//		E_WorkingStates.NOTIFY_LOADING_OUTBOUND:
//			ton_timeout.PT	:= T#1S;
//			///////////////there is no tote in working position/////////////
//			IF NOT(roller_inbound.photo_sensor[0].Q OR roller_inbound.photo_sensor[1].Q OR photo_sensor_tote_detection.Q OR roller_outbound.photo_sensor.Q) THEN
//				IF sInstanceName='working1' THEN
//					subData.Topic	:= E_Topics.LOADING_BEGIN_OUTBOUND_WOKING1;
//					GVL.PubSubService.Publish(topic:=E_Topics.LOADING_BEGIN_OUTBOUND_WOKING1,data:= subData);				
//				END_IF
//				IF sInstanceName='working2' THEN
//					subData.Topic	:= E_Topics.LOADING_BEGIN_OUTBOUND_WOKING2;
//					GVL.PubSubService.Publish(topic:=E_Topics.LOADING_BEGIN_OUTBOUND_WOKING2,data:= subData);				
//				END_IF
//				eStates	:= E_WorkingStates.WAIT_NEW_TOTE;
//			END_IF	
//			///////////////there is a tote in working position/////////////
//			IF NOT roller_inbound.photo_sensor[0].Q AND roller_inbound.photo_sensor[1].Q AND photo_sensor_tote_detection.Q AND NOT roller_outbound.photo_sensor.Q THEN
//				eStates	:= E_WorkingStates.BAG_OPEN_DOWN;
//			END_IF					
			
		E_WorkingStates.WAIT_NEW_TOTE:	
			///////////////there is a tote in working position/////////////
			IF NOT roller_inbound.photo_sensor[0].Q AND roller_inbound.photo_sensor[1].Q AND photo_sensor_tote_detection.Q AND NOT roller_outbound.photo_sensor.Q THEN
				eStates	:= E_WorkingStates.BAG_OPEN_DOWN;
			END_IF			
		/////////////////////////abort inbound command from app///////////////////
			IF xAbortInbound THEN
				xAbortInbound	:= FALSE;
				tote_status	:= ToteStatus.VACANT;
				M_load	:= TRUE;
				eStates	:= E_WorkingStates.IDLE;				
			ELSE
				tote_status	:= ToteStatus.AWAITING_INBOUND_AVAILABILITY;
			END_IF
		//////////////////////////normal process///////////////////////
			IF sInstanceName='working1' THEN
				IF xBeginInbound AND GVL.fb_loading.valve_left_door.retracted THEN
					xBeginInbound	:=FALSE;
					eStates	:= E_WorkingStates.WAIT_MUTE_SENSOR_ON;
				END_IF					
			END_IF
			IF sInstanceName='working2' THEN
				IF xBeginInbound AND GVL.fb_loading.valve_right_door.retracted THEN
					xBeginInbound	:=FALSE;
					eStates	:= E_WorkingStates.WAIT_MUTE_SENSOR_ON;
				END_IF					
			END_IF
		/////////////////////////////while in stopping/////////////////////			
			IF  THIS^.eState = ePMLState_Stopping THEN
				IF sInstanceName='working1' THEN//publish to loading for loading might be not in stopping
					subData.Topic	:= E_Topics.LOADING_END_OUTBOUND_WOKING1;
					GVL.PubSubService.Publish(topic:=E_Topics.LOADING_END_OUTBOUND_WOKING1,data:= subData);				
				END_IF
				IF sInstanceName='working2' THEN
					subData.Topic	:= E_Topics.LOADING_END_OUTBOUND_WOKING2;
					GVL.PubSubService.Publish(topic:=E_Topics.LOADING_END_OUTBOUND_WOKING2,data:= subData);				
				END_IF
				M_load	:= TRUE;
				eStates	:= E_WorkingStates.IDLE;
			END_IF						
////////////////////////////////////////////////action/////////////////////////////////////////////
			
		E_WorkingStates.WAIT_MUTE_SENSOR_ON:	
			tote_status	:= ToteStatus.INBOUNDING;
			ton_timeout.PT	:= T#2S;	
			roller_inbound.roller.forward	:= TRUE;
			IF  roller_inbound.photo_sensor[0].Q THEN
				eStates	:= E_WorkingStates.WAIT_TOTE_DETECTION_ON;
			END_IF			
		E_WorkingStates.WAIT_TOTE_DETECTION_ON:
			roller_inbound.roller.forward	:= TRUE;
			IF photo_sensor_tote_detection.Q THEN
				eStates	:= E_WorkingStates.WAIT_MUTE_SENSOR_OFF;
			END_IF
		E_WorkingStates.WAIT_MUTE_SENSOR_OFF:
			roller_inbound.roller.forward	:= TRUE;
			IF NOT roller_inbound.photo_sensor[0].Q THEN
				eStates	:= E_WorkingStates.WAIT_LOAD_SENSOR_ON;
			END_IF
		E_WorkingStates.WAIT_LOAD_SENSOR_ON:
			roller_inbound.roller.forward	:= TRUE;
			IF roller_inbound.photo_sensor[1].Q THEN	
				roller_inbound.roller.forward	:= FALSE;
				eStates	:= E_WorkingStates.BAG_OPEN_DOWN;
			END_IF
		E_WorkingStates.BAG_OPEN_DOWN:
			st_mcAxis_lift.mcMoveAbsolute.Execute	:= TRUE;		
			st_mcAxis_lift.rActualPosSet	:= rPos_lift_down;
			st_mcAxis_lift.rVelocitySet	:= 250;
			IF st_mcAxis_lift.mcMoveAbsolute.Done THEN	
				eStates	:= E_WorkingStates.BAG_OPEN;
			END_IF		
		E_WorkingStates.BAG_OPEN:	
			ton_timeout.PT	:= T#3S;		
			st_mcAxis_bag.mcMoveAbsolute.Execute	:= TRUE;		
			st_mcAxis_bag.rActualPosSet	:= rPos_bag_opened;
			st_mcAxis_bag.rVelocitySet	:= 50;
			IF st_mcAxis_bag.mcMoveAbsolute.Done OR st_mcAxis_bag.bTouchTorque THEN			
				st_mcAxis_bag.mcMoveAbsolute.Execute	:= FALSE;
				eStates	:= E_WorkingStates.BAG_OPEN_DETECTION;
			END_IF	
		E_WorkingStates.BAG_OPEN_DETECTION:	
			IF ABS(st_mcAxis_bag.rActualPos-rPos_bag_opened)>5 THEN
				bagOpen_Status[0].bag_status	:= BagStatus.ERROR;
				bagOpen_Status[1].bag_status	:= BagStatus.ERROR;
				tote_status	:= ToteStatus.BAG_OPEN_FAILED;
				eStates	:= E_WorkingStates.DONE;
				RETURN;
			END_IF
			ton_timeout.PT	:= INT_TO_TIME(iDelay_sensor_detection);
			IF ton_timeout.Q THEN
				/////////////////////////////////////////////bag openner1/////////////////////////////////////////					
				FOR i:=0 TO 3 DO
					IF BagOpening_Detection[i] THEN
						bagOpen_Status[0].sensor_status	:=CONCAT(STR1:=bagOpen_Status[0].sensor_status,STR2:='1');
						bagOpen_Status[0].iCnt_sensor_detection	:=bagOpen_Status[0].iCnt_sensor_detection+1;
					ELSE
						bagOpen_Status[0].sensor_status	:=CONCAT(STR1:=bagOpen_Status[0].sensor_status,STR2:='0');
					END_IF
				END_FOR	
				IF bagOpen_Status[0].iCnt_sensor_detection>=iSensor_detection_setting[0] THEN
					bagOpen_Status[0].bag_status	:= BagStatus.OPENED;
					strLog_bagopen_detection	:= CONCAT(STR1:=bag_opening_status[0].sensor_status,STR2:='->OPENED;');
				ELSE
					bagOpen_Status[0].bag_status	:= BagStatus.ERROR;
					strLog_bagopen_detection	:= CONCAT(STR1:=bag_opening_status[0].sensor_status,STR2:='->ERROR;');
				END_IF			
				/////////////////////////////////////////////bag openner2/////////////////////////////////////////	
				FOR i:=4 TO 7 DO
					IF BagOpening_Detection[i] THEN
						bagOpen_Status[1].sensor_status	:=CONCAT(STR1:=bagOpen_Status[1].sensor_status,STR2:='1');
						bagOpen_Status[1].iCnt_sensor_detection	:=bagOpen_Status[1].iCnt_sensor_detection+1;
					ELSE
						bagOpen_Status[1].sensor_status	:=CONCAT(STR1:=bagOpen_Status[1].sensor_status,STR2:='0');
					END_IF
				END_FOR		
				IF bagOpen_Status[1].iCnt_sensor_detection>=iSensor_detection_setting[1] THEN
					bagOpen_Status[1].bag_status	:= BagStatus.OPENED;
					strLog_bagopen_detection	:= CONCAT(STR1:=bag_opening_status[1].sensor_status,STR2:='->OPENED');
				ELSE
					bagOpen_Status[1].bag_status	:= BagStatus.ERROR;
					strLog_bagopen_detection	:= CONCAT(STR1:=bag_opening_status[1].sensor_status,STR2:='->ERROR');
				END_IF				

	
				eStates	:= E_WorkingStates.TOTE_STATUS_DETECTION;	
			END_IF
		E_WorkingStates.TOTE_STATUS_DETECTION:
			IF bUsingOpenBag THEN
				IF bagOpen_Status[0].bag_status=BagStatus.OPENED AND bagOpen_Status[1].bag_status=BagStatus.OPENED THEN
					tote_status	:= ToteStatus.LOADED;
				ELSE
					tote_status	:= ToteStatus.BAG_OPEN_FAILED;
				END_IF
			ELSE
				tote_status	:= ToteStatus.LOADED;
			END_IF
			/////////////////////////////////////////writelog////////////////////////////////////////
			IF bagOpen_Status[0].bag_status=BagStatus.OPENED THEN
				strLog_bagopen_detection	:= CONCAT(STR1:=bagOpen_Status[0].sensor_status,STR2:='->OPENED;');
			ELSE	
				strLog_bagopen_detection	:= CONCAT(STR1:=bagOpen_Status[0].sensor_status,STR2:='->ERROR;');
			END_IF
			IF bagOpen_Status[1].bag_status=BagStatus.OPENED THEN
				strLog_bagopen_detection	:= CONCAT(STR1:=strLog_bagopen_detection,STR2:=bagOpen_Status[1].sensor_status);
				strLog_bagopen_detection	:= CONCAT(STR1:=strLog_bagopen_detection,STR2:='->OPENED;');
			ELSE	
				strLog_bagopen_detection	:= CONCAT(STR1:=strLog_bagopen_detection,STR2:=bagOpen_Status[1].sensor_status);
				strLog_bagopen_detection	:= CONCAT(STR1:=strLog_bagopen_detection,STR2:='->ERROR;');
			END_IF					
			eStates	:= E_WorkingStates.DONE;		
		E_WorkingStates.DONE:
			ADSLOGSTR(msgCtrlMask:= ADSLOG_MSGTYPE_LOG,msgFmtStr:=strLog_bagopen_detection,strArg:='');
			M_load	:= TRUE;
			eStates	:= E_WorkingStates.IDLE;
			

		
		
END_CASE
END_METHOD

METHOD M_mapping : BOOL
VAR_INPUT
END_VAR
IF sInstanceName='working1' THEN
	
	/////////////////////////////////////digital input-2024.5.25////////////////////////////////////////

	roller_inbound.roller.err(D:= G_IO.arDI[4].Ch[0],on_ms:=500,off_ms:=80);	
	roller_inbound.photo_sensor[0](D:= arIOLinkQualifier_Place1.CH[3].1,on_ms:=200,off_ms:=300);  //入口料框检测
	roller_inbound.photo_sensor[1](D:= arIOLinkQualifier_Place1.CH[3].0,on_ms:=100,off_ms:=100);  //X向到位感应
	
	roller_outbound.roller.err(D:= G_IO.arDI[4].Ch[1],on_ms:=500,off_ms:=80);	
	roller_outbound.photo_sensor(D:= arIOLinkQualifier_Place1.CH[4].0,on_ms:=100,off_ms:=80);   //Y向出料口感应

	roller_outbound_assist.roller.err(D:= G_IO.arDI[4].Ch[2],on_ms:=500,off_ms:=80);	
	EDM_KM            							:= G_IO.arDI[4].Ch[3];       //P24_sto反馈  
				  
	photo_sensor_tote_detection(D:= arIOLinkQualifier_Place1.CH[4].1,on_ms:=100,off_ms:=100);  //XY对角料框感应
		
	BagOpening_Detection[0]:= arIOLinkTx_Place1[7].	InputByte[1].0;
	BagOpening_Detection[1]:= arIOLinkTx_Place1[7].	InputByte[0].0;
	BagOpening_Detection[2]:= arIOLinkTx_Place1[7].	InputByte[1].1;
	BagOpening_Detection[3]:= arIOLinkTx_Place1[7].	InputByte[0].1;
	BagOpening_Detection[4]:= arIOLinkTx_Place1[7].	InputByte[1].2;
	BagOpening_Detection[5]:= arIOLinkTx_Place1[7].	InputByte[0].2;
	BagOpening_Detection[6]:= arIOLinkTx_Place1[7].	InputByte[1].3;
	BagOpening_Detection[7]:= arIOLinkTx_Place1[7].	InputByte[0].3;
		
	valve_lift.extended		:= arIOLinkQualifier_Place1.CH[0].1 AND arIOLinkQualifier_Place1.CH[1].1;
	valve_lift.retracted	:= arIOLinkQualifier_Place1.CH[2].1 AND arIOLinkQualifier_Place1.CH[2].0;
		
	(****************************axis_lift*******************************************************)
		
	st_mcAxis_lift.limit_sensor_positive:= arIOLinkQualifier_Place1.CH[5].0	 ;
	st_mcAxis_lift.limit_sensor_negative:= arIOLinkQualifier_Place1.CH[5].1  ;
	st_mcAxis_lift.limit_sensor_home	:= arIOLinkQualifier_Place1.CH[6].1  ;
		
		
		
		
	(****************************axis_bagopener***************************************************)
	st_mcAxis_bag.limit_sensor_positive:= 	arIOLinkTx_Place1[7].InputByte[0].4 ;
	st_mcAxis_bag.limit_sensor_negative:= 	arIOLinkTx_Place1[7].InputByte[0].5 ;
	//using software limit position for
		
		
		
		
		
	/////////////////////////////////////digital output-2024.5.25////////////////////////////////////////
	G_IO.arDO[6].Ch[0]	:= valve_lift.extend;
	G_IO.arDO[6].Ch[1]	:= valve_lift.retract;
		
	G_IO.arDO[4].Ch[2]	:= roller_inbound.roller.forward;
	G_IO.arDO[4].Ch[3]	:= roller_inbound.roller.backward;		
	G_IO.arDO[4].Ch[4]	:= roller_outbound.roller.backward;
	G_IO.arDO[4].Ch[5]	:= roller_outbound.roller.forward;		
	G_IO.arDO[4].Ch[6]	:= roller_outbound_assist.roller.forward;
	G_IO.arDO[4].Ch[7]	:= roller_outbound_assist.roller.backward;
			
	/////////////////////////////////////axis config////////////////////////////////////////
	mcAxis_lift
	(
		ZSN		:=   st_mcAxis_lift.limit_sensor_negative OR st_mcAxis_lift.xHoming, //TODO link to digital input
		ZSP		:=   st_mcAxis_lift.limit_sensor_positive  OR st_mcAxis_lift.xHoming, //TODO link to digital input
		IN_OUT	:= st_mcAxis_lift	, 
		AXIS	:= AxisRef_lift	, 
	);
	st_mcAxis_lift.bPosSensorShow	:= TRUE;
	st_mcAxis_lift.bNegSensorShow	:= TRUE;
	st_mcAxis_lift.bStopButtonShow	:= TRUE;
	st_mcAxis_lift.rMaxAcceleration	:= 50000;
	st_mcAxis_lift.rMaxDeceleration	:= 50000;
	st_mcAxis_lift.rMaxJerk			:= 500000;
	st_mcAxis_lift.rAcceleration	:= 2500;
	st_mcAxis_lift.rDeceleration	:= 2500;
	st_mcAxis_lift.rJerk			:= 12500;
	st_mcAxis_lift.rMaxVelocity		:= 100;
	st_mcAxis_lift.rMaxDistance		:= 50;
	st_mcAxis_lift.bPosSen	:=  st_mcAxis_lift.limit_sensor_positive ;//TODO link to digital input
	st_mcAxis_lift.bNegSen	:=  st_mcAxis_lift.limit_sensor_negative ;//TODO link to digital input
	st_mcAxis_lift.mcHome.bCalibrationCam	:= TRUE;//TODO link to digital input origin
	st_mcAxis_lift.bPositionSensor	:= TRUE;//TODO link to digital input origin
	st_mcAxis_lift.bdirFW	:= TRUE;
	st_mcAxis_lift.sNetID := '192.168.17.27.6.1';
	st_mcAxis_lift.nSlaveAddr	:= 1009;
	st_mcAxis_lift.rToqueLimitSet	:= 80;
		
	mcAxis_bag
	(
		ZSN		:=   st_mcAxis_bag.limit_sensor_negative OR st_mcAxis_bag.xHoming, //TODO link to digital input
		ZSP		:=   st_mcAxis_bag.limit_sensor_positive OR st_mcAxis_bag.xHoming, //TODO link to digital input
		IN_OUT	:= st_mcAxis_bag	, 
		AXIS	:= AxisRef_bag	, 
	);
	st_mcAxis_bag.bPosSensorShow	:= TRUE;
	st_mcAxis_bag.bNegSensorShow	:= TRUE;
	st_mcAxis_bag.bStopButtonShow	:= TRUE;
	st_mcAxis_bag.rMaxAcceleration	:= 50000;
	st_mcAxis_bag.rMaxDeceleration	:= 50000;
	st_mcAxis_bag.rMaxJerk			:= 500000;
	st_mcAxis_bag.rAcceleration	:= 500;
	st_mcAxis_bag.rDeceleration	:= 500;
	st_mcAxis_bag.rJerk			:= 2000;
	st_mcAxis_bag.rMaxVelocity		:= 300;
	st_mcAxis_bag.rMaxDistance		:= 50;
	st_mcAxis_bag.bPosSen	:=  st_mcAxis_bag.limit_sensor_positive ;//TODO link to digital input
	st_mcAxis_bag.bNegSen	:=  st_mcAxis_bag.limit_sensor_negative ;//TODO link to digital input
	st_mcAxis_bag.mcHome.bCalibrationCam	:= TRUE;//TODO link to digital input origin
	st_mcAxis_bag.bPositionSensor	:= TRUE;//TODO link to digital input origin
	st_mcAxis_bag.bdirFW	:= TRUE;
	st_mcAxis_bag.sNetID := '192.168.17.27.6.1';
	st_mcAxis_bag.nSlaveAddr	:= 1010;
	st_mcAxis_bag.rToqueLimitSet	:= 80;
	st_mcAxis_bag.rToqueSet	:= 25;
		//st_mcAxis_bag.rActTorque	:= actTorque;
//		st_mcAxis_bag.bTouque_control_enable	:=ABS(st_mcAxis_bag.rActualPos-rPos_bag_opened)>10 AND xLoading;
		
		rPos_bag_closed_step_0	:= rPos_bag_opened-rPos_bag_preopen;
END_IF
IF sInstanceName='working2' THEN
	/////////////////////////////////////digital input-2024.5.25////////////////////////////////////////

	roller_inbound.roller.err(D:= G_IO.arDI[6].Ch[0],on_ms:=500,off_ms:=80); 
	roller_inbound.photo_sensor[0](D:= arIOLinkQualifier_Place2.CH[3].1,on_ms:=100,off_ms:=80);  //入口料框检测
	roller_inbound.photo_sensor[1](D:= arIOLinkQualifier_Place2.CH[3].0,on_ms:=100,off_ms:=80);  //X向到位感应
	
	roller_outbound.roller.err(D:= G_IO.arDI[6].Ch[1],on_ms:=500,off_ms:=80); 
	roller_outbound.photo_sensor(D:= arIOLinkQualifier_Place2.CH[4].0,on_ms:=100,off_ms:=80);   //Y向出料口感应
	
	roller_outbound_assist.roller.err(D:= G_IO.arDI[6].Ch[2],on_ms:=500,off_ms:=80); 
	EDM_KM            							:= G_IO.arDI[6].Ch[3];       //P24_sto反馈  
			  
	photo_sensor_tote_detection(D:= arIOLinkQualifier_Place2.CH[4].1,on_ms:=100,off_ms:=100);  //XY对角料框感应
	
	BagOpening_Detection[0]:= arIOLinkTx_Place2[7].	InputByte[1].0;
	BagOpening_Detection[1]:= arIOLinkTx_Place2[7].	InputByte[0].0;
	BagOpening_Detection[2]:= arIOLinkTx_Place2[7].	InputByte[1].1;
	BagOpening_Detection[3]:= arIOLinkTx_Place2[7].	InputByte[0].1;
	BagOpening_Detection[4]:= arIOLinkTx_Place2[7].	InputByte[1].2;
	BagOpening_Detection[5]:= arIOLinkTx_Place2[7].	InputByte[0].2;
	BagOpening_Detection[6]:= arIOLinkTx_Place2[7].	InputByte[1].3;
	BagOpening_Detection[7]:= arIOLinkTx_Place2[7].	InputByte[0].3;
	
	
	valve_lift.extended     := arIOLinkQualifier_Place2.CH[0].1 AND arIOLinkQualifier_Place2.CH[2].1;
	valve_lift.retracted    := arIOLinkQualifier_Place2.CH[1].1 AND arIOLinkQualifier_Place2.CH[2].0 ;
	
	(****************************axis_lift*******************************************************)
	
	st_mcAxis_lift.limit_sensor_positive:=  arIOLinkQualifier_Place2.CH[5].0;
	st_mcAxis_lift.limit_sensor_negative:=  arIOLinkQualifier_Place2.CH[5].1;
	st_mcAxis_lift.limit_sensor_home:= 		arIOLinkQualifier_Place2.CH[6].1;
	
	(****************************axis_bagopener***************************************************)
	st_mcAxis_bag.limit_sensor_positive	:= arIOLinkTx_Place2[7].	InputByte[0].4 ;
	st_mcAxis_bag.limit_sensor_negative	:= arIOLinkTx_Place2[7].	InputByte[0].5 ;
	st_mcAxis_bag.limit_sensor_home		:= arIOLinkTx_Place2[7].	InputByte[1].5 ;
	
	
	/////////////////////////////////////digital output-2024.5.25////////////////////////////////////////
	G_IO.arDO[7].Ch[0]	:= valve_lift.extend;
	G_IO.arDO[7].Ch[1]	:= valve_lift.retract;
	
	G_IO.arDO[5].Ch[2]	:= roller_inbound.roller.forward;
	G_IO.arDO[5].Ch[3]	:= roller_inbound.roller.backward;	
	G_IO.arDO[5].Ch[4]	:= roller_outbound.roller.forward;
	G_IO.arDO[5].Ch[5]	:= roller_outbound.roller.backward;
	G_IO.arDO[5].Ch[6]	:= roller_outbound_assist.roller.forward;
	G_IO.arDO[5].Ch[7]	:= roller_outbound_assist.roller.backward;
	
	/////////////////////////////////////axis config////////////////////////////////////////
	mcAxis_lift
	(
		ZSN		:=   st_mcAxis_lift.limit_sensor_negative OR st_mcAxis_lift.xHoming, //TODO link to digital input
		ZSP		:=   st_mcAxis_lift.limit_sensor_positive OR st_mcAxis_lift.xHoming, //TODO link to digital input
		IN_OUT	:= st_mcAxis_lift	, 
		AXIS	:= AxisRef_lift	, 
	);
	st_mcAxis_lift.bPosSensorShow	:= TRUE;
	st_mcAxis_lift.bNegSensorShow	:= TRUE;
	st_mcAxis_lift.bStopButtonShow	:= TRUE;
	st_mcAxis_lift.rMaxAcceleration	:= 50000;
	st_mcAxis_lift.rMaxDeceleration	:= 50000;
	st_mcAxis_lift.rMaxJerk			:= 500000;
	st_mcAxis_lift.rAcceleration	:= 2500;
	st_mcAxis_lift.rDeceleration	:= 2500;
	st_mcAxis_lift.rJerk			:= 12500;
	st_mcAxis_lift.rMaxVelocity		:= 100;
	st_mcAxis_lift.rMaxDistance		:= 50;
	st_mcAxis_lift.bPosSen	:=  st_mcAxis_lift.limit_sensor_positive ;//TODO link to digital input
	st_mcAxis_lift.bNegSen	:=  st_mcAxis_lift.limit_sensor_negative ;//TODO link to digital input
	st_mcAxis_lift.mcHome.bCalibrationCam	:= TRUE;//TODO link to digital input origin
	st_mcAxis_lift.bPositionSensor	:= TRUE;//TODO link to digital input origin
	st_mcAxis_lift.bdirFW	:= TRUE;
	st_mcAxis_lift.sNetID := '192.168.17.27.7.1';
	st_mcAxis_lift.nSlaveAddr	:= 1009;
	st_mcAxis_lift.rToqueLimitSet	:= 80;
	
	mcAxis_bag
	(
		ZSN		:=   st_mcAxis_bag.limit_sensor_negative OR st_mcAxis_bag.xHoming, //TODO link to digital input
		ZSP		:=   st_mcAxis_bag.limit_sensor_positive OR st_mcAxis_bag.xHoming, //TODO link to digital input
		IN_OUT	:= st_mcAxis_bag	, 
		AXIS	:= AxisRef_bag	, 
	);
	st_mcAxis_bag.bPosSensorShow	:= TRUE;
	st_mcAxis_bag.bNegSensorShow	:= TRUE;
	st_mcAxis_bag.bStopButtonShow	:= TRUE;
	st_mcAxis_bag.rMaxAcceleration	:= 50000;
	st_mcAxis_bag.rMaxDeceleration	:= 50000;
	st_mcAxis_bag.rMaxJerk			:= 500000;
	st_mcAxis_bag.rAcceleration	:= 500;
	st_mcAxis_bag.rDeceleration	:= 500;
	st_mcAxis_bag.rJerk			:= 2000;
	st_mcAxis_bag.rMaxVelocity		:= 300;
	st_mcAxis_bag.rMaxDistance		:= 50;
	st_mcAxis_bag.bPosSen	:=  st_mcAxis_bag.limit_sensor_positive ;//TODO link to digital input
	st_mcAxis_bag.bNegSen	:=  st_mcAxis_bag.limit_sensor_negative ;//TODO link to digital input
	st_mcAxis_bag.mcHome.bCalibrationCam	:= TRUE;//TODO link to digital input origin
	st_mcAxis_bag.bPositionSensor	:= TRUE;//TODO link to digital input origin
	st_mcAxis_bag.bdirFW	:= TRUE;
	st_mcAxis_bag.sNetID := '192.168.17.27.7.1';
	st_mcAxis_bag.nSlaveAddr	:= 1010;
	st_mcAxis_bag.rToqueLimitSet	:= 80;
	st_mcAxis_bag.rToqueSet	:= 25;
	//st_mcAxis_bag.rActTorque	:= actTorque;
	//st_mcAxis_bag.bTouque_control_enable	:=ABS(st_mcAxis_bag.rActualPos-rPos_bag_opened)>10 AND xLoading;
	
	rPos_bag_closed_step_0	:= rPos_bag_opened-8;

END_IF
END_METHOD

METHOD M_Reset
VAR_INPUT
END_VAR
//Take away all commands
IF GVL.stChangeIntoProduction.bYesReset THEN
;
END_IF
END_METHOD

{attribute 'object_name' := 'M_Resetting'}
METHOD M_Resetting
CASE fbUnitModeManager.eModeStatus OF
	ePMLProtUnitMode_Production:		//Production, Mantainance, Manual
		valve_lift.extend	:= FALSE;
		valve_lift.retract	:= TRUE;
		st_mcAxis_lift.mcStop.Execute	:= FALSE;
		st_mcAxis_bag.mcStop.Execute	:= FALSE;
		st_mcAxis_lift.mcReset.Execute			:= TRUE;
		st_mcAxis_bag.mcReset.Execute			:= TRUE;		
		error_status	:= OrderToteErrorStatus.NO_ERROR;	
		ton_timeout.IN	:= FALSE;
		M_StateComplete();
	
	ePMLProtUnitMode_Maintenance, ePMLProtUnitMode_Manual, ePMLUnitMode_Service:
		M_StateComplete();
END_CASE
END_METHOD

{attribute 'object_name' := 'M_Starting'}
METHOD M_Starting
CASE fbUnitModeManager.eModeStatus OF
	ePMLProtUnitMode_Production:		//Production, Mantainance, Manual
		ton_timeout.IN	:=FALSE;
		st_mcAxis_bag.mcPower.Enable	:= TRUE;
		st_mcAxis_lift.mcPower.Enable	:= TRUE;
		IF logtech_control_command=LogTechControlCmd.TRANSFER_TOTE_FINISHED THEN		
			logtech_control_command	:= LogTechControlCmd.DO_NOTHING;	
		END_IF
		IF M_checkCondition(condition:=E_Condition.TOTE_READY) THEN
			IF tote_status = ToteStatus.LOADED OR tote_status = ToteStatus.VACANT THEN
				eStates	:= E_WorkingStates.IDLE;
				xInbound	:= FALSE;
				xOutbound	:= FALSE;
			END_IF
			IF tote_status=ToteStatus.MECHANICAL_ERROR THEN
				IF xInbound THEN
					tote_status	:= ToteStatus.INBOUNDING;
				END_IF
				IF xOutbound THEN
					tote_status	:= ToteStatus.OUTBOUNDING;
				END_IF
			END_IF			
			IF st_mcAxis_bag.mcPower.Status AND st_mcAxis_lift.mcPower.Status THEN
				M_StateComplete();
			END_IF
		END_IF
		
		
	ePMLProtUnitMode_Maintenance, ePMLProtUnitMode_Manual, ePMLUnitMode_Service:
		M_StateComplete();
END_CASE
END_METHOD

{attribute 'object_name' := 'M_Stopping'}
METHOD M_Stopping
CASE fbUnitModeManager.eModeStatus OF
	ePMLProtUnitMode_Production, ePMLProtUnitMode_Manual:
/////////////////////////////////////////////////////////	
		IF NOT xInbound AND NOT xOutbound THEN
			M_StateComplete();
			RETURN;
		END_IF
//////////////////////////unloading///////////////////////	
		IF xOutbound THEN	
			IF M_unload() THEN
			 	xOutbound := FALSE;						
				M_StateComplete();
			END_IF	
			RETURN;
		END_IF	
//////////////////////////loading///////////////////////
		IF xInbound THEN
			IF PreviousState=ePMLState_Idle THEN
				M_StateComplete();
				RETURN;	
			END_IF
				
			IF M_load() THEN
				xInbound	:= FALSE;						
				M_StateComplete();
			END_IF
		END_IF		
	

				
	ePMLProtUnitMode_Maintenance, ePMLUnitMode_Service:
		M_StateComplete();	
			//not defined
END_CASE
END_METHOD

{attribute 'object_name' := 'M_Undefined'}
METHOD M_Undefined

bUndefinedDone					:= TRUE;
END_METHOD

METHOD M_unload : BOOL
VAR_INPUT
END_VAR

M_unload := FALSE;
//event.sMethod	:= 'unload';

//////////////////////////////////////////////////////////timeout//////////////////////////////////////////
		iStateTemp	:= eStateTemp;
//		ton_timeout();
		IF eStateTemp=eStates THEN
			ton_timeout.IN	:=TRUE;
		ELSE
			ton_timeout.IN	:=FALSE;
			eStateTemp	:= eStates;	
			M_Log(eLogType:=ServerityLevelType.INFO,sTextLog:='');
			IF ton_timeout.Q THEN
				RETURN;
			END_IF
		END_IF
		IF ton_timeout.Q THEN	
			ton_timeout.IN	:=FALSE;
			CASE eStates OF	
				E_LoadingStates.ERROR:	
					alarm_temp.Message	:= GenerateErrorMsg(errorType:='M',iState := iStateTemp,errorMsg:='in error state.');
				ELSE
					alarm_temp.Message	:= GenerateErrorMsg(errorType:='M',iState := iStateTemp,errorMsg:='time out');
			END_CASE
//////////////////////////////////////////////////////////states don't want to timeout and trig error//////////////////////////////////////////				
			IF  eStates<>E_WorkingStates.IDLE AND 
				eStates<>E_WorkingStates.WAIT_UNLOADING AND 
				eStates<>E_WorkingStates.BAG_OPEN_UP AND
				eStates<>E_WorkingStates.WAIT_LOGTECH_OUTBOUND 
			THEN
				IF sInstanceName='working1' THEN
					tote_status	:= ToteStatus.MECHANICAL_ERROR;	
					THIS^.pml_adminAlarm.M_SetAlarm(stAdmin:=GVL.PackTags1.Admin,stAlarm:=THIS^.alarm_temp);					
				END_IF
				IF sInstanceName='working2' THEN
					tote_status	:= ToteStatus.MECHANICAL_ERROR;	
					THIS^.pml_adminAlarm.M_SetAlarm(stAdmin:=GVL.PackTags2.Admin,stAlarm:=THIS^.alarm_temp);					
				END_IF						

			END_IF
		END_IF
		

CASE eStates OF 
		E_WorkingStates.IDLE:
			st_mcAxis_lift.mcReset.Execute	:= TRUE;
			st_mcAxis_bag.mcReset.Execute	:= TRUE;			
			IF ton_timeout.Q THEN
				eStates	:= E_WorkingStates.INIT;
			END_IF		
		E_WorkingStates.INIT:	
			ton_timeout.PT	:= T#3S;
			bagOpen_Status	:= bagOpenInit_Status;			
			st_mcAxis_lift.mcMoveAbsolute.Execute	:= FALSE;
			st_mcAxis_bag.mcMoveAbsolute.Execute	:= FALSE;
			IF M_checkCondition(condition:=E_Condition.TOTE_READY) THEN///////////check tote status
				IF tote_status=ToteStatus.VACANT THEN
					eStates	:= E_WorkingStates.DONE;
				ELSE
					eStates	:= E_WorkingStates.WAIT_UNLOADING;
				END_IF
			END_IF		
		E_WorkingStates.WAIT_UNLOADING://wait signal from logtech and app to unload the tote
			logtech_status	:= LogTechStatus.RUNNING;//todo:remove while on site
			IF logtech_status=LogTechStatus.RUNNING THEN
				tote_status	:= ToteStatus.AWAITING_OUTBOUND_AVAILABILITY;
				IF bUsingOpenBag THEN
					eStates	:= E_WorkingStates.BAG_CLOSE_STEP_0;
				ELSE
					eStates	:= E_WorkingStates.BAG_OPEN_UP;
				END_IF				
			ELSE
				tote_status	:= ToteStatus.DOWNSTREAM_NOT_READY;
			END_IF	
		E_WorkingStates.BAG_CLOSE_STEP_0:
			IF error_status=OrderToteErrorStatus.BAG_OPEN_FAILED THEN
				st_mcAxis_bag.mcMoveAbsolute.Execute	:= TRUE;		
				st_mcAxis_bag.rActualPosSet	:= rPos_bag_closed;
				st_mcAxis_bag.rVelocitySet	:= 250;				
			ELSE
				IF NOT (ABS(st_mcAxis_bag.rActualPos-rPos_bag_closed_step_0)<0.1) THEN
					st_mcAxis_bag.mcMoveAbsolute.Execute	:= TRUE;		
					st_mcAxis_bag.rActualPosSet	:= rPos_bag_closed_step_0;
					st_mcAxis_bag.rVelocitySet	:= 250;				
				END_IF
			END_IF
			IF st_mcAxis_bag.mcMoveAbsolute.Done OR (ABS(st_mcAxis_bag.rActualPos-rPos_bag_closed_step_0)<0.1) THEN
				st_mcAxis_bag.mcMoveAbsolute.Execute	:= FALSE;
				eStates	:= E_WorkingStates.BAG_OPEN_UP;
			END_IF	
		E_WorkingStates.BAG_OPEN_UP:
			ton_timeout.PT	:= T#3S;
			IF bRobot_in_safety_place THEN		
				st_mcAxis_lift.mcMoveAbsolute.Execute	:= TRUE;		
				st_mcAxis_lift.rActualPosSet	:= rPos_lift_up;
				st_mcAxis_lift.rVelocitySet	:= 250;
				IF st_mcAxis_lift.mcMoveAbsolute.Done THEN
					st_mcAxis_lift.mcMoveAbsolute.Execute	:= FALSE;
					eStates	:= E_WorkingStates.TOTE_LIFT_UP;
				END_IF	
			END_IF
		E_WorkingStates.TOTE_LIFT_UP:
			valve_lift.extend	:= TRUE;
			valve_lift.retract	:= FALSE;
			IF valve_lift.extended AND NOT valve_lift.retracted THEN
				eStates	:= E_WorkingStates.WAIT_LOGTECH_OUTBOUND;
			END_IF										
		E_WorkingStates.WAIT_LOGTECH_OUTBOUND:			
			/////////////////////////abort outbound command from app///////////////////
			IF xAbortOutbound THEN
				xAbortOutbound	:= FALSE;
				tote_status	:= ToteStatus.LOADED;
				outboundTote_status	:= ToteStatus.VACANT;
				M_unload	:= TRUE;
				eStates	:= E_WorkingStates.IDLE;				
			ELSE
			//////////////////////////normal process///////////////////////
				tote_status	:= ToteStatus.AWAITING_OUTBOUND_AVAILABILITY;
				outboundTote_status	:= ToteStatus.AWAITING_INBOUND_AVAILABILITY;
				logtech_control_command	:= LogTechControlCmd.READY_TO_TRANSFER;
				logtech_transfer_status	:= LogTechTransferStatus.READY_TO_RECEIVE;//todo:remove while onsite
				IF logtech_transfer_status=LogTechTransferStatus.READY_TO_RECEIVE THEN
					eStates	:= E_WorkingStates.TOTE_UNLOAD;
				END_IF	
			END_IF			
			/////////////////////////////while in stopping/////////////////////	
			IF  eState = ePMLState_Stopping THEN
				tote_status	:= ToteStatus.LOADED;
				outboundTote_status	:= ToteStatus.VACANT;
				M_unload	:= TRUE;
				xOutbound	:= FALSE;
				eStates	:= E_WorkingStates.IDLE;
			END_IF
		E_WorkingStates.TOTE_UNLOAD:
			tote_status	:= ToteStatus.OUTBOUNDING;
			outboundTote_status	:= ToteStatus.INBOUNDING;
			logtech_control_command	:= LogTechControlCmd.TRANSFERRING_TOTE;
			valve_lift.extend	:= TRUE;
			valve_lift.retract	:= FALSE;		
			ton_timeout.PT	:= T#2S;
			roller_outbound.roller.forward		:= TRUE;
			roller_outbound_assist.roller.forward	:= TRUE;
			IF roller_outbound.photo_sensor.Q THEN
				eStates	:= E_WorkingStates.WAIT_TOTE_DETECTION_OFF;			
			END_IF	
		E_WorkingStates.WAIT_TOTE_DETECTION_OFF:	
			valve_lift.extend	:= TRUE;
			valve_lift.retract	:= FALSE;				
			roller_outbound.roller.forward		:= TRUE;
			roller_outbound_assist.roller.forward	:= TRUE;
			IF NOT photo_sensor_tote_detection.Q THEN
				eStates	:= E_WorkingStates.WAIT_SENSOR_OFF;	
			END_IF
		E_WorkingStates.WAIT_SENSOR_OFF:
			valve_lift.extend	:= TRUE;
			valve_lift.retract	:= FALSE;		
			roller_outbound.roller.forward		:= TRUE;
			roller_outbound_assist.roller.forward	:= TRUE;	
			IF NOT roller_outbound.photo_sensor.Q THEN
				eStates	:= E_WorkingStates.WAIT_RECEIVE_TOTE_FINISHED;			
			END_IF			
		E_WorkingStates.WAIT_RECEIVE_TOTE_FINISHED:
			valve_lift.extend	:= TRUE;
			valve_lift.retract	:= FALSE;			
			roller_outbound.roller.forward		:= TRUE;
			roller_outbound_assist.roller.forward	:= TRUE;
			logtech_control_command	:= LogTechControlCmd.TRANSFER_TOTE_FINISHED;
			logtech_transfer_status	:= LogTechTransferStatus.RECEIVE_TOTE_FINISHED;//todo:remove while onsite
			IF	logtech_transfer_status=LogTechTransferStatus.RECEIVE_TOTE_FINISHED THEN
				roller_outbound.roller.forward		:= FALSE;	
				roller_outbound_assist.roller.forward	:= FALSE;
				logtech_control_command	:= LogTechControlCmd.DO_NOTHING;
				eStates	:= E_WorkingStates.TOTE_LIFT_DOWN;
			END_IF
		E_WorkingStates.TOTE_LIFT_DOWN:
			roller_outbound.roller.forward		:= FALSE;	
			roller_outbound_assist.roller.forward	:= FALSE;	
			st_mcAxis_bag.mcMoveAbsolute.Execute	:= TRUE;		
			st_mcAxis_bag.rVelocitySet	:= 250;
			IF bUsingOpenBag THEN
				st_mcAxis_bag.rActualPosSet	:= rPos_bag_closed;
			ELSE
				st_mcAxis_bag.rActualPosSet	:= rPos_bag_opened;
			END_IF
			valve_lift.extend	:= FALSE;
			valve_lift.retract	:= TRUE;
			IF st_mcAxis_bag.mcMoveAbsolute.Done AND NOT valve_lift.extended AND valve_lift.retracted THEN
				st_mcAxis_bag.mcMoveAbsolute.Execute	:= FALSE;
				eStates	:= E_WorkingStates.DONE;
			END_IF				
		E_WorkingStates.DONE:	
			logtech_control_command	:= LogTechControlCmd.DO_NOTHING;
			tote_status	:= ToteStatus.VACANT;
			outboundTote_status	:= ToteStatus.LOADED;		
			M_unload	:= TRUE;
			eStates	:= E_WorkingStates.IDLE;



		
END_CASE
END_METHOD

METHOD M_waitCondition : BOOL
VAR_INPUT
	condition	: E_Condition;
END_VAR
M_waitCondition	:= FALSE;
CASE condition OF
	E_Condition.NO_TOTE:
	 	IF NOT roller_inbound.photo_sensor[1].Q THEN
			M_waitCondition	:= TRUE;
		END_IF
	E_Condition.TOTE_IN:
	 	IF roller_inbound.photo_sensor[1].Q THEN
			M_waitCondition	:= TRUE;
		END_IF	
	E_Condition.READY_LOADING_TOTE:
		IF  GVL.fb_loading.eTransfer=E_Transfer.UNLOAD
			OR tote_status=ToteStatus.LOADED 
			OR  xInbound
		THEN
			M_waitCondition	:= TRUE;
		END_IF	
END_CASE
END_METHOD

METHOD ParseStateToString : STRING
VAR_INPUT
END_VAR
CASE THIS^.eStates OF
	E_WorkingStates.IDLE:
		ParseStateToString	:='IDLE';
	E_WorkingStates.INIT:
		ParseStateToString	:='INIT';
	E_WorkingStates.CHECK:
		ParseStateToString	:='CHECK';
	E_WorkingStates.WAIT_NEW_TOTE:
		ParseStateToString	:='WAIT_NEW_TOTE';
	E_WorkingStates.LOADING:
		ParseStateToString	:='LOADING';
	E_WorkingStates.WAIT_FINISHED:
		ParseStateToString	:='WAIT_FINISHED';
	E_WorkingStates.TOTE_LOAD:
		ParseStateToString	:='TOTE_LOAD';
	E_WorkingStates.TOTE_UNLOAD:
		ParseStateToString	:='TOTE_UNLOAD';
	E_WorkingStates.BAG_OPEN:
		ParseStateToString	:='BAG_OPEN';
	E_WorkingStates.BAG_OPEN_DETECTION:
		ParseStateToString	:='BAG_OPEN_DETECTION';
	E_WorkingStates.BAG_CLOSE_STEP_0:
		ParseStateToString	:='BAG_CLOSE_STEP_0';
	E_WorkingStates.BAG_CLOSE_STEP_1:
		ParseStateToString	:='BAG_CLOSE_STEP_1';
	E_WorkingStates.BAG_CLOSE:
		ParseStateToString	:='BAG_CLOSE';
	E_WorkingStates.BAG_OPEN_INIT:
		ParseStateToString	:='BAG_OPEN_INIT';
	E_WorkingStates.TOTE_LIFT_UP:
		ParseStateToString	:='TOTE_LIFT_UP';
	E_WorkingStates.TOTE_LIFT_DOWN:
		ParseStateToString	:='TOTE_LIFT_DOWN';
	E_WorkingStates.BAG_OPEN_UP:
		ParseStateToString	:='BAG_OPEN_UP';
	E_WorkingStates.BAG_OPEN_DOWN:
		ParseStateToString	:='BAG_OPEN_DOWN';
	E_WorkingStates.TOTE_OUT:
		ParseStateToString	:='TOTE_OUT';
	E_WorkingStates.WAIT_1:
		ParseStateToString	:='WAIT_1';
	E_WorkingStates.WAIT_LOGTECH_OUTBOUND:
		ParseStateToString	:='WAIT_LOGTECH_OUTBOUND';
	E_WorkingStates.TOTE_STATUS_DETECTION:
		ParseStateToString	:='TOTE_STATUS_DETECTION';
	E_WorkingStates.NOTIFY_LOADING_OUTBOUND:
		ParseStateToString	:='NOTIFY_LOADING_OUTBOUND';
	E_WorkingStates.AGING_STATE_0:
		ParseStateToString	:='AGING_STATE_0';
	E_WorkingStates.AGING_STATE_1:
		ParseStateToString	:='AGING_STATE_1';
	E_WorkingStates.WAIT:
		ParseStateToString	:='WAIT';
	E_WorkingStates.WAIT_UNLOADING:
		ParseStateToString	:='WAIT_UNLOADING';
	E_WorkingStates.WAIT_SENSOR_ON:
		ParseStateToString	:='WAIT_SENSOR_ON';
	E_WorkingStates.WAIT_SENSOR_OFF:
		ParseStateToString	:='WAIT_SENSOR_OFF';
	E_WorkingStates.WAIT_MUTE_SENSOR_ON:
		ParseStateToString	:='WAIT_MUTE_SENSOR_ON';
	E_WorkingStates.WAIT_MUTE_SENSOR_OFF:
		ParseStateToString	:='WAIT_MUTE_SENSOR_OFF';
	E_WorkingStates.WAIT_LOAD_SENSOR_ON:
		ParseStateToString	:='WAIT_LOAD_SENSOR_ON';
	E_WorkingStates.WAIT_LOAD_SENSOR_OFF:
		ParseStateToString	:='WAIT_LOAD_SENSOR_OFF';
	E_WorkingStates.WAIT_RECEIVE_TOTE_FINISHED:
		ParseStateToString	:='WAIT_RECEIVE_TOTE_FINISHED';
	E_WorkingStates.WAIT_TOTE_DETECTION_ON:
		ParseStateToString	:='WAIT_TOTE_DETECTION_ON';
	E_WorkingStates.WAIT_TOTE_DETECTION_OFF:
		ParseStateToString	:='WAIT_TOTE_DETECTION_OFF';
	E_WorkingStates.DONE:
		ParseStateToString	:='DONE';
	E_WorkingStates.ERROR:
		ParseStateToString	:='ERROR';
	ELSE
		ParseStateToString	:='UNKNOW STATE';
END_CASE
END_METHOD

END_FUNCTION_BLOCK

// ---- Ads/Ads/BagOpeningStatus.TcPOU
FUNCTION_BLOCK BagOpeningStatus
VAR_INPUT
END_VAR
VAR_OUTPUT
END_VAR
VAR
	bag_status	: BagStatus;
	sensor_status	: STRING;
END_VAR

PROPERTY _bagStatus : BagStatus
GET
_bagStatus	:= bag_status;
END_GET
SET
bag_status	:= _bagStatus;
END_SET
END_PROPERTY

PROPERTY _sensor_status : STRING
GET
_sensor_status	:= sensor_status;
END_GET
SET
sensor_status	:=_sensor_status;
END_SET
END_PROPERTY

END_FUNCTION_BLOCK

// ---- PubSub/PubSubService.TcPOU
FUNCTION_BLOCK PubSubService IMPLEMENTS I_PubSubService
VAR_INPUT
END_VAR
VAR_OUTPUT
END_VAR

VAR
	TopicsToSubscribers : ARRAY[0..MAX_TOPICS - 1, 0..MAX_SUBSCRIBERS_PER_TOPIC - 1] OF SubscriberCell;
	subscriberCounters : ARRAY [0..MAX_TOPICS - 1] OF INT;
	cntPublish	: ST_TracePublish;
END_VAR

VAR CONSTANT 
	MAX_SUBSCRIBERS_PER_TOPIC : INT := 5;
	MAX_TOPICS : INT := E_Topics.NUMBER_OF_TOPICS;
END_VAR

METHOD ParseStateToString : STRING
VAR_INPUT
	topic	: E_Topics;
END_VAR
CASE topic OF
	E_Topics.UNKNOWN:
		ParseStateToString	:='UNKNOWN';
	E_Topics.WORKING1_INBOUND_TOTE:
		ParseStateToString	:='WORKING1_INBOUND_TOTE';
	E_Topics.WORKING1_OUTBOUND_TOTE:
		ParseStateToString	:='WORKING1_OUTBOUND_TOTE';
	E_Topics.LOADING_BEGIN_OUTBOUND_WOKING1:
		ParseStateToString	:='LOADING_BEGIN_OUTBOUND_WOKING1';
	E_Topics.LOADING_END_OUTBOUND_WOKING1:
		ParseStateToString	:='LOADING_END_OUTBOUND_WOKING1';
	E_Topics.WORKING1_BEGIN_INBOUND:
		ParseStateToString	:='WORKING1_BEGIN_INBOUND';
	E_Topics.WORKING1_ABORT_INBOUND:
		ParseStateToString	:='WORKING1_ABORT_INBOUND';
	E_Topics.WORKING2_INBOUND_TOTE:
		ParseStateToString	:='WORKING2_INBOUND_TOTE';
	E_Topics.WORKING2_OUTBOUND_TOTE:
		ParseStateToString	:='WORKING2_OUTBOUND_TOTE';
	E_Topics.LOADING_BEGIN_OUTBOUND_WOKING2:
		ParseStateToString	:='LOADING_BEGIN_OUTBOUND_WOKING2';
	E_Topics.LOADING_END_OUTBOUND_WOKING2:
		ParseStateToString	:='LOADING_END_OUTBOUND_WOKING2';
	E_Topics.WORKING2_BEGIN_INBOUND:
		ParseStateToString	:='WORKING2_BEGIN_INBOUND';
	E_Topics.WORKING2_ABORT_INBOUND:
		ParseStateToString	:='WORKING2_ABORT_INBOUND';	
	E_Topics.RESET_WAITING_FOR_NEW_SPACE:
		ParseStateToString	:='RESET_WAITING_FOR_NEW_SPACE';				
	E_Topics.SAMPLE_SUBSCRRIBE_1:
		ParseStateToString	:='SAMPLE_SUBSCRRIBE_1';	
	E_Topics.SAMPLE_SUBSCRRIBE_2:
		ParseStateToString	:='SAMPLE_SUBSCRRIBE_2';	
	E_Topics.SAMPLE_SUBSCRRIBE_3:
		ParseStateToString	:='SAMPLE_SUBSCRRIBE_3';	
	E_Topics.NUMBER_OF_TOPICS:
		ParseStateToString	:='NUMBER_OF_TOPICS';		
		
	ELSE
		ParseStateToString	:='UNKNOW TOPIC';
END_CASE
END_METHOD

METHOD Publish
VAR_INPUT
	topic	: E_Topics;
	data	: PubSubData;
END_VAR
VAR
	index : INT;
END_VAR
cntPublish.iCnt	:= 0;
cntPublish.topic	:= '';	
FOR index := 0 TO MAX_SUBSCRIBERS_PER_TOPIC -1 BY 1 DO
	IF TopicsToSubscribers[topic, index].OCCUPIED = TRUE THEN
		TopicsToSubscribers[topic, index].subscriber.Callback(data);
//		ADSLOGSTR(msgCtrlMask:=Tc2_System.ADSLOG_MSGTYPE_LOG,msgFmtStr:=CONCAT(STR1:=ParseStateToString(topic),STR2:=TopicsToSubscribers[topic, index].sInstance),strArg:='');
	END_IF
	cntPublish.iCnt		:= cntPublish.iCnt+1;
	cntPublish.topic	:= ParseStateToString(topic);	
END_FOR
END_METHOD

METHOD Subscribe : INT
VAR_INPUT
	topic	: E_Topics;
	sInstance	: STRING;
	subCallback	: I_SubCallback;
END_VAR
VAR 
	index : INT;
END_VAR
Subscribe := -1;

IF  subscriberCounters[topic] >= MAX_SUBSCRIBERS_PER_TOPIC THEN
	RETURN;
END_IF

FOR index := 0 TO (MAX_SUBSCRIBERS_PER_TOPIC - 1) BY 1 DO
	IF TopicsToSubscribers[topic, index].occupied = FALSE THEN
		TopicsToSubscribers[topic, index].occupied := TRUE;
		TopicsToSubscribers[topic, index].sTopic := ParseStateToString(topic);
		TopicsToSubscribers[topic, index].sInstance := sInstance;
		TopicsToSubscribers[topic, index].subscriber := subCallback;
		Subscribe := index;
		subscriberCounters[topic] := subscriberCounters[topic] + 1;
		RETURN;
	END_IF
END_FOR
END_METHOD

METHOD Unsubscribe
VAR_INPUT
	topic : E_Topics;
	subscriberID	: INT;
END_VAR
IF TopicsToSubscribers[topic, subscriberID].occupied = TRUE THEN
	TopicsToSubscribers[topic, subscriberID].occupied := FALSE;
	subscriberCounters[topic] := subscriberCounters[topic] - 1; 	
END_IF
END_METHOD

END_FUNCTION_BLOCK

// ---- Mian/FB_autoStore.TcPOU
FUNCTION_BLOCK FB_autoStore EXTENDS FB_Generic
VAR_INPUT
END_VAR
VAR_OUTPUT
END_VAR
VAR
	lamp			: BOOL;	
	eStates			: E_AutoStore_States := E_AutoStore_States.IDLE;;
	eStateTemp		: E_AutoStore_States := E_AutoStore_States.IDLE;
	
	mcAxis_lift 			: FB_MotionAxis_MC;
	st_mcAxis_lift 			: ST_MotionAxis_MC;
	AxisRef_lift			: AXIS_REF;
	
	mcAxis_transfer 		: FB_MotionAxis_MC;
	st_mcAxis_transfer		: ST_MotionAxis_MC;
	AxisRef_transfer		: AXIS_REF;
	
	door_closed						: BOOL;
	button_start					: BOOL;	
	button_stop						: BOOL;	
	sensor_lift_atDownPos			: BOOL;
	sensor_transfer_atWorkingPos	: BOOL;
	sensor_transfer_atFeedingPos	: BOOL;
	
	bUpStairs						: BOOL;
	bExchangeTote					: BOOL;
END_VAR	
VAR PERSISTENT
	rPos_lift_up				: REAL;
	rPos_lift_down				: REAL;
	rPos_transfer_feeding		: REAL;
	rPos_transfer_working		: REAL;	
END_VAR

SUPER^();

IF sInstanceName='autoStore_1' THEN
	IF NOT subscribed THEN
		GVL.PubSubService.Subscribe(E_Topics.AUTOSTORE1_EXCHANGE,sInstanceName,THIS^);
		subscribed	:= TRUE;
	END_IF
END_IF
IF sInstanceName='autoStore_2' THEN
	IF NOT subscribed THEN
		GVL.PubSubService.Subscribe(E_Topics.AUTOSTORE2_EXCHANGE,sInstanceName,THIS^);
		subscribed	:= TRUE;
	END_IF
END_IF


//sComponent_name		:= _sInstanceName;
//iComponetID			:= ModuleID.SAMPLE1;

infoLevel	:= ServerityLevelType.WARNING;

(*
Description: 
the callback that will be invoked when there is a publish for what the subscriber was subscribed to.
*)
METHOD Callback
VAR_INPUT
	data : PubSubData;
END_VAR

IF sInstanceName='autoStore_1' THEN
	CASE data.Topic OF
		E_Topics.AUTOSTORE1_EXCHANGE:
			bExchangeTote	:= TRUE;		
	END_CASE	
END_IF
IF sInstanceName='autoStore_2' THEN
	CASE data.Topic OF
		E_Topics.AUTOSTORE2_EXCHANGE:
			bExchangeTote	:= TRUE;		
	END_CASE	
END_IF
END_METHOD

{attribute 'object_name' := 'M_Aborting'}
METHOD M_Aborting
CASE fbUnitModeManager.eModeStatus OF	
	ePMLProtUnitMode_Production, ePMLProtUnitMode_Manual:		

		st_mcAxis_lift.mcMoveAbsolute.Execute		:= FALSE;
		st_mcAxis_lift.mcStop.Execute				:= TRUE;	
		st_mcAxis_transfer.mcMoveAbsolute.Execute	:= FALSE;
		st_mcAxis_transfer.mcStop.Execute			:= TRUE;
		iAging_test	:= 0;
		M_StateComplete();
			
	ePMLProtUnitMode_Maintenance, ePMLUnitMode_Service:
		
		M_StateComplete();
END_CASE
END_METHOD

METHOD M_agingTest : BOOL
VAR_INPUT
	rVelocity_percent	: REAL;
END_VAR
END_METHOD

{attribute 'object_name' := 'M_Completing'}
METHOD M_Completing
CASE fbUnitModeManager.eModeStatus OF
	ePMLProtUnitMode_Production:
		;
END_CASE
END_METHOD

{attribute 'object_name' := 'M_Execute'}
METHOD M_Execute

CASE fbUnitModeManager.eModeStatus OF
	ePMLProtUnitMode_Production:		//Mode Production
//////////////////////////////////////////////////////////timeout//////////////////////////////////////////	
		iStateTemp	:= eStateTemp;
		ton_timeout();
		IF eStateTemp=eStates THEN
			ton_timeout.IN	:=TRUE;
		ELSE
			ton_timeout.IN	:=FALSE;
			eStateTemp	:= eStates;	
			M_Log(eLogType:=ServerityLevelType.INFO,sTextLog:='');
			IF ton_timeout.Q THEN
				RETURN;
			END_IF
		END_IF
		IF ton_timeout.Q THEN	
			ton_timeout.IN	:=FALSE;
			CASE eStates OF	
				E_AutoStore_States.ERROR:	
					alarm_temp.Message	:= GenerateErrorMsg(errorType:='M',iState := iStateTemp,errorMsg:='in error state.');
				ELSE
				alarm_temp.Message	:= GenerateErrorMsg(errorType:='M',iState := iStateTemp,errorMsg:='time out');
			END_CASE
//////////////////////////////////////////////////////////states don't want to timeout and trig error//////////////////////////////////////////				
			IF 	eStates<>E_AutoStore_States.IDLE AND
				eStates<>E_AutoStore_States.WAIT AND
				eStates<>E_AutoStore_States.WAIT_CMD
			THEN 
				IF sInstanceName='autoStore_1' THEN
					GVL.pml_adminAlarm.M_SetAlarm(stAdmin:=GVL.PackTags1.Admin,stAlarm:=alarm_temp);
				END_IF
				IF sInstanceName='autoStore_2' THEN
					GVL.pml_adminAlarm.M_SetAlarm(stAdmin:=GVL.PackTags2.Admin,stAlarm:=alarm_temp);
				END_IF					
			END_IF
		END_IF
//////////////////////////////////////////////////////////auto running process//////////////////////////////////////////			
		CASE eStates OF 
				E_AutoStore_States.IDLE:
					ton_timeout.PT	:= T#1MS;						
					eStates	:= E_AutoStore_States.INIT;				
				E_AutoStore_States.INIT:
					ton_timeout.PT	:= T#1S;
					eStates	:= E_AutoStore_States.WAIT; 
				E_AutoStore_States.WAIT:
					ton_timeout.PT	:= T#10S;
					eStates	:= E_AutoStore_States.WAIT_CMD; 
				E_AutoStore_States.WAIT_CMD:
					IF bExchangeTote THEN
						bExchangeTote	:= FALSE;
						eStates	:= E_AutoStore_States.LIFT_MOVE_DOWN;
					END_IF
				////////////////////////////lift move down///////////////////////////////////		
				E_AutoStore_States.LIFT_MOVE_DOWN:	
					st_mcAxis_lift.mcMoveAbsolute.Execute	:= TRUE;					
					st_mcAxis_lift.rActualPosSet	:= rPos_lift_down;
					st_mcAxis_lift.rVelocitySet		:= 100;					
					IF st_mcAxis_lift.mcMoveAbsolute.Done THEN
						eStates	:= E_AutoStore_States.LIFT_DOWN_SENSOR_DETECTED;
					END_IF
				E_AutoStore_States.LIFT_DOWN_SENSOR_DETECTED:	
					IF sensor_lift_atDownPos THEN
						IF bUpStairs THEN
							eStates	:= E_AutoStore_States.TRANSFER_MOVE_FEEDING;
							bUpStairs	:= FALSE;
						ELSE
							eStates	:= E_AutoStore_States.TRANSFER_MOVE_WORKING;
							bUpStairs	:= TRUE;
						END_IF					
					END_IF
				////////////////////////////upstairs///////////////////////////////////	
				E_AutoStore_States.TRANSFER_MOVE_FEEDING:	
					st_mcAxis_transfer.mcMoveAbsolute.Execute	:= TRUE;					
					st_mcAxis_transfer.rActualPosSet	:= rPos_transfer_feeding;
					st_mcAxis_transfer.rVelocitySet		:= 100;					
					IF st_mcAxis_transfer.mcMoveAbsolute.Done THEN
						eStates	:= E_AutoStore_States.TRANSFER_FEEDING_SENSOR_DETECTED;
					END_IF				

				E_AutoStore_States.TRANSFER_FEEDING_SENSOR_DETECTED:
					IF sensor_transfer_atFeedingPos OR TRUE THEN//todo:add this sensor
						eStates	:= E_AutoStore_States.LIFT_MOVE_UP;
					END_IF									
				////////////////////////////downstairs///////////////////////////////////		
				E_AutoStore_States.TRANSFER_MOVE_WORKING:	
					st_mcAxis_transfer.mcMoveAbsolute.Execute	:= TRUE;					
					st_mcAxis_transfer.rActualPosSet	:= rPos_transfer_working;
					st_mcAxis_transfer.rVelocitySet		:= 100;					
					IF st_mcAxis_transfer.mcMoveAbsolute.Done THEN
						eStates	:= E_AutoStore_States.TRANSFER_WORKING_SENSOR_DETECTED;
					END_IF					
				E_AutoStore_States.TRANSFER_WORKING_SENSOR_DETECTED:
					IF sensor_transfer_atWorkingPos THEN
						eStates	:= E_AutoStore_States.LIFT_MOVE_UP;
					END_IF
					
				////////////////////////////lift move up///////////////////////////////////	
				E_AutoStore_States.LIFT_MOVE_UP:
					st_mcAxis_lift.mcMoveAbsolute.Execute	:= TRUE;					
					st_mcAxis_lift.rActualPosSet	:= rPos_lift_up;
					st_mcAxis_lift.rVelocitySet		:= 100;					
					IF st_mcAxis_lift.mcMoveAbsolute.Done THEN
						eStates	:= E_AutoStore_States.DONE;
					END_IF		

				
				E_AutoStore_States.DONE:
					eStates	:= E_AutoStore_States.IDLE;
				E_AutoStore_States.ERROR:
					;
			END_CASE
		
		
	ePMLProtUnitMode_Maintenance, ePMLUnitMode_Service:		
		//
		
	ePMLProtUnitMode_Manual:		//Manaul

END_CASE
END_METHOD

{attribute 'object_name' := 'M_Holding'}
METHOD M_Holding
CASE fbUnitModeManager.eModeStatus OF
	ePMLProtUnitMode_Production:		//Mode Production
		//Finisch the actual seperationstep	
		

	ePMLProtUnitMode_Maintenance:
		M_StateComplete();
END_CASE
END_METHOD

{attribute 'object_name' := 'M_Idle'}
METHOD M_Idle
IF G_HMI.bAging_test THEN
	//M_agingTest();
END_IF
END_METHOD

METHOD M_mapping : BOOL
VAR_INPUT
END_VAR

		
		
		
	(****************************digital input***************************************************)
	st_mcAxis_lift.limit_sensor_positive		:= 	arDI[20].Ch[0] ;
	st_mcAxis_lift.limit_sensor_negative		:= 	arDI[20].Ch[1] ;
	door_closed									:= 	arDI[20].Ch[2] ;
	button_start								:= 	arDI[20].Ch[3] ;
	button_stop									:= 	arDI[20].Ch[4] ;
	sensor_lift_atDownPos						:= 	arDI[20].Ch[5] ;
	st_mcAxis_transfer.limit_sensor_positive	:= 	arDI[20].Ch[6] ;
	st_mcAxis_transfer.limit_sensor_negative	:= 	arDI[20].Ch[7] ;	
	sensor_transfer_atWorkingPos				:= 	arDI[20].Ch[8] ;	
//	sensor_transfer_atFeedingPos				:= 	arDI[20].Ch[9] ;	
		

	/////////////////////////////////////axis config////////////////////////////////////////
	mcAxis_lift
	(
		ZSN		:=   st_mcAxis_lift.limit_sensor_negative OR st_mcAxis_lift.xHoming, //TODO link to digital input
		ZSP		:=   (st_mcAxis_lift.limit_sensor_positive AND sensor_transfer_atWorkingPos)  OR st_mcAxis_lift.xHoming, //TODO link to digital input
		IN_OUT	:= st_mcAxis_lift	, 
		AXIS	:= AxisRef_lift	, 
	);
	st_mcAxis_lift.bPosSensorShow	:= TRUE;
	st_mcAxis_lift.bNegSensorShow	:= TRUE;
	st_mcAxis_lift.bStopButtonShow	:= TRUE;
	st_mcAxis_lift.rMaxAcceleration	:= 50000;
	st_mcAxis_lift.rMaxDeceleration	:= 50000;
	st_mcAxis_lift.rMaxJerk			:= 500000;
	st_mcAxis_lift.rAcceleration	:= 2500;
	st_mcAxis_lift.rDeceleration	:= 2500;
	st_mcAxis_lift.rJerk			:= 12500;
	st_mcAxis_lift.rMaxVelocity		:= 100;
	st_mcAxis_lift.rMaxDistance		:= 50;
	st_mcAxis_lift.bPosSen	:=  st_mcAxis_lift.limit_sensor_positive ;//TODO link to digital input
	st_mcAxis_lift.bNegSen	:=  st_mcAxis_lift.limit_sensor_negative ;//TODO link to digital input
	st_mcAxis_lift.mcHome.bCalibrationCam	:= TRUE;//TODO link to digital input origin
	st_mcAxis_lift.bPositionSensor	:= TRUE;//TODO link to digital input origin
	st_mcAxis_lift.bdirFW	:= TRUE;
	st_mcAxis_lift.sNetID := '192.168.17.27.6.1';
	st_mcAxis_lift.nSlaveAddr	:= 1009;
	st_mcAxis_lift.rToqueLimitSet	:= 80;
	
	mcAxis_transfer
	(
		ZSN		:=   (st_mcAxis_transfer.limit_sensor_negative AND sensor_lift_atDownPos) OR st_mcAxis_transfer.xHoming, //TODO link to digital input
		ZSP		:=   (st_mcAxis_transfer.limit_sensor_positive AND sensor_lift_atDownPos) OR st_mcAxis_transfer.xHoming, //TODO link to digital input
		IN_OUT	:= st_mcAxis_transfer	, 
		AXIS	:= AxisRef_transfer	, 
	);
	st_mcAxis_transfer.bPosSensorShow	:= TRUE;
	st_mcAxis_transfer.bNegSensorShow	:= TRUE;
	st_mcAxis_transfer.bStopButtonShow	:= TRUE;
	st_mcAxis_transfer.rMaxAcceleration	:= 50000;
	st_mcAxis_transfer.rMaxDeceleration	:= 50000;
	st_mcAxis_transfer.rMaxJerk			:= 500000;
	st_mcAxis_transfer.rAcceleration	:= 2500;
	st_mcAxis_transfer.rDeceleration	:= 2500;
	st_mcAxis_transfer.rJerk			:= 12500;
	st_mcAxis_transfer.rMaxVelocity		:= 100;
	st_mcAxis_transfer.rMaxDistance		:= 50;
	st_mcAxis_transfer.bPosSen	:=  st_mcAxis_transfer.limit_sensor_positive ;//TODO link to digital input
	st_mcAxis_transfer.bNegSen	:=  st_mcAxis_transfer.limit_sensor_negative ;//TODO link to digital input
	st_mcAxis_transfer.mcHome.bCalibrationCam	:= TRUE;//TODO link to digital input origin
	st_mcAxis_transfer.bPositionSensor	:= TRUE;//TODO link to digital input origin
	st_mcAxis_transfer.bdirFW	:= TRUE;
	st_mcAxis_transfer.sNetID := '192.168.17.27.6.1';
	st_mcAxis_transfer.nSlaveAddr	:= 1009;
	st_mcAxis_transfer.rToqueLimitSet	:= 80;
END_METHOD

METHOD M_Reset
VAR_INPUT
END_VAR
//Take away all commands
IF GVL.stChangeIntoProduction.bYesReset THEN
;
END_IF
END_METHOD

{attribute 'object_name' := 'M_Resetting'}
METHOD M_Resetting
CASE fbUnitModeManager.eModeStatus OF
	ePMLProtUnitMode_Production:		//Production, Mantainance, Manual
		lamp	:= FALSE;
		eStates :=E_SampleStates.IDLE;
		M_StateComplete();
	
	ePMLProtUnitMode_Maintenance, ePMLProtUnitMode_Manual, ePMLUnitMode_Service:
		M_StateComplete();
END_CASE
END_METHOD

{attribute 'object_name' := 'M_Starting'}
METHOD M_Starting
CASE fbUnitModeManager.eModeStatus OF
	ePMLProtUnitMode_Production:		//Production, Mantainance, Manual
		
		M_StateComplete();
	ePMLProtUnitMode_Maintenance, ePMLProtUnitMode_Manual, ePMLUnitMode_Service:
		M_StateComplete();
END_CASE
END_METHOD

{attribute 'object_name' := 'M_Stopping'}
METHOD M_Stopping
CASE fbUnitModeManager.eModeStatus OF
	ePMLProtUnitMode_Production, ePMLProtUnitMode_Manual:
				//////////////////////////////////////////////////////////timeout//////////////////////////////////////////	
		iStateTemp	:= eStateTemp;
		ton_timeout();
		IF eStateTemp=eStates THEN
			ton_timeout.IN	:=TRUE;
		ELSE
			ton_timeout.IN	:=FALSE;
			eStateTemp	:= eStates;	
		END_IF
		IF ton_timeout.Q THEN	
			ton_timeout.IN	:=FALSE;
			CASE eStates OF		
				E_SampleStates.IDLE:						
					;
				E_SampleStates.INIT:
					;
				E_SampleStates.WAIT_ON:
					;
				E_SampleStates.WAIT_OFF:
					;			
				E_SampleStates.ERROR:	
					alarm_temp.Message	:= 'Sample in error state';
				ELSE
					alarm_temp.Message	:= 'UNKNOWN STATES in Sample module';
			END_CASE
			IF eStates<>E_SampleStates.IDLE AND eStates<>E_SampleStates.WAIT_ON AND eStates<>E_SampleStates.WAIT_OFF THEN
				GVL.pml_adminAlarm.M_SetAlarm(stAdmin:=GVL.PackTags.Admin,stAlarm:=alarm_temp);
			END_IF
		END_IF
		
		CASE eStates OF 
				E_SampleStates.IDLE:						
					eStates	:= E_SampleStates.INIT;				
				E_SampleStates.INIT:
					ton_timeout.PT	:= T#1S;
					eStates	:= E_SampleStates.WAIT_ON; 
				E_SampleStates.WAIT_ON:
					lamp	:= TRUE;
					IF ton_timeout.Q THEN
						eStates	:= E_SampleStates.WAIT_OFF;
					END_IF
				E_SampleStates.WAIT_OFF:
					lamp	:= FALSE;
					IF ton_timeout.Q THEN
						eStates	:= E_SampleStates.IDLE;
						M_StateComplete();	
					END_IF
				E_SampleStates.ERROR:
					;
			END_CASE			
	ePMLProtUnitMode_Maintenance, ePMLUnitMode_Service:
		M_StateComplete();	
			//not defined
END_CASE
END_METHOD

{attribute 'object_name' := 'M_Undefined'}
METHOD M_Undefined

bUndefinedDone					:= TRUE;
END_METHOD

METHOD ParseStateToString : STRING
VAR_INPUT
END_VAR
CASE THIS^.eStates OF
	E_AutoStore_States.IDLE:
		ParseStateToString	:='IDLE';
	E_AutoStore_States.INIT:
		ParseStateToString	:='INIT';
	E_AutoStore_States.CHECK:
		ParseStateToString	:='CHECK';

	E_AutoStore_States.WAIT:
		ParseStateToString	:='WAIT';

	E_AutoStore_States.DONE:	
		ParseStateToString	:='DONE';
	E_AutoStore_States.ERROR:
		ParseStateToString	:='ERROR';
	ELSE
		ParseStateToString	:='UNKNOW STATE';
END_CASE
END_METHOD

END_FUNCTION_BLOCK

// ---- Ads/FB_MachineControl_Subsystem.TcPOU
FUNCTION_BLOCK FB_MachineControl_Subsystem
VAR_INPUT
	pMachineCurrentStatus	:POINTER TO E_PMLState;
END_VAR
VAR_OUTPUT
END_VAR
VAR
	machine_status AT%Q*: MachineStatus:= MachineStatus.STOPPED;	
	machine_current_status	: E_PMLState;	
    machineControlCmd	: MachineCommandStructure;
	
	

	bStart	: BOOL;
	bStop	: BOOL;
	bReset	: BOOL;
	machineControlCmd_temp	: MachineCommandStructure;
	AAA: INT;
END_VAR


CASE pMachineCurrentStatus^ OF
	ePMLState_Stopped:
		machine_status	:= MachineStatus.STOPPED;
	ePMLState_Resetting:	
		machine_status	:= MachineStatus.RESETTING;
	ePMLState_Idle:	
		machine_status	:= MachineStatus.READY;	
	ePMLState_Starting:	
		machine_status	:= MachineStatus.INITIALIZING;
	ePMLState_Execute:	
		machine_status	:= MachineStatus.RUNNING;		
	ePMLState_Stopping:	
		machine_status	:= MachineStatus.STOPPING;
	ePMLState_Aborted,ePMLState_Aborting:
		machine_status	:= MachineStatus.ERROR;		
END_CASE




IF bStart THEN
	machineControlCmd_temp.command	:= MachineControlCommand.START;
	machine_control_command(command_data:=machineControlCmd_temp);
	bStart	:= FALSE;
END_IF
IF bStop THEN
	machineControlCmd_temp.command	:= MachineControlCommand.STOP;
	machine_control_command(command_data:=machineControlCmd_temp);
	bStop	:= FALSE;
END_IF
IF bReset THEN
	machineControlCmd_temp.command	:= MachineControlCommand.RESET;
	machine_control_command(command_data:=machineControlCmd_temp);
	bReset	:= FALSE;
END_IF

{attribute 'TcRpcEnable'}
METHOD machine_control_command : UDINT
VAR_INPUT
	command_data : MachineCommandStructure; 	
END_VAR

machineControlCmd	:= command_data;
AAA:=AAA+1;
END_METHOD

END_FUNCTION_BLOCK

// ---- Ads/FB_Safety_Subsystem.TcPOU
FUNCTION_BLOCK FB_Safety_Subsystem EXTENDS FB_Generic
VAR_INPUT
	pHeartBeat		: POINTER TO FB_HeartBeat_Subsystem;
	pSafety_door	: POINTER TO ST_safetyDoor;
	pPackTags		: POINTER TO ST_PackMLv30;
	pMachine		: POINTER TO FB_Machine;
END_VAR
VAR_IN_OUT
	
END_VAR
VAR_OUTPUT
	
END_VAR
VAR
	button_array AT%Q* : ARRAY [0..99] OF ButtonStatus; (* Array of 100 elements for ButtonStatus, button reset, button unlock *)
	estop_array AT%Q* : ARRAY [0..99] OF EStopStatus; (* Array of 100 elements for EStopStatus *)
	safety_door_array AT%Q*: ARRAY [0..99] OF SafetyDoorStatus; (* Array of 100 elements for SafetyDoorStatus *)
	light_curtain_array AT%Q*: ARRAY [0..999] OF LightCurtainStatus; (* Array of 1000 elements for LightCurtainStatus *)
	sensor_array  AT%Q*: ARRAY [0..999] OF SensorStatus; (* Array of 1000 elements for SensorStatus *)
	estop_status AT%Q*: GeneralStatus;
	gates_status AT%Q*: GeneralStatus;
	safety_status AT%Q*: GeneralStatus;

	SI_0	: UINT;
	SI_1	: UINT;
	GI_0 	: UINT;
	GI_1 	: UINT;
	
	
	station_mode	: StationMode;//APP status
	iStationMode	: UINT;
	iState: INT;
	bEstop_detection	: BOOL;	
	

	eStates					:	E_SafetyStates	:=	E_SafetyStates.IDLE;
	eStateTemp				:	E_SafetyStates	:=	E_SafetyStates.IDLE;

	errorMessage	: STRING;
	xError	: BOOL;
	xEstop	: BOOL;
	xError_working	: BOOL;
	xEstop_behavior	: BOOL;
	
	xError_loading	: BOOL;
	eStates_safetyDoor	: E_SAFETYDOOR	:= E_SAFETYDOOR.IDLE;
	bReset_safetyDoor	: BOOL;
	
	
	
	GPWM	: FB_GPWM;
	GPWM_1s	: FB_GPWM;
	tonSaftyDelay: TON;
	b_EStopRestarting  : BOOL;
	T_EStopRestart : TON;
//////////////////////SAFETY hardware config///////////////	
	mcp_estop_left				: FB_DigitalInput;
	safetyDoor_left				: BOOL;
	
	mcp_estop_right				: FB_DigitalInput;
	safetyDoor_right			: BOOL;
	door_closed					: BOOL;
	bRobot1_eStop				: BOOL;
	bRobot2_eStop				: BOOL;

	lift_station_detection		: BOOL;
	
	lift_door_left				: FB_DigitalInput;
	lift_door_right				: FB_DigitalInput;
	
	robot1_EES					: BOOL;
	robot1_EAS					: BOOL;
	
	robot2_EES					: BOOL;
	robot2_EAS					: BOOL;
	buffer_safety				: BOOL;
	loading_safety				: BOOL;
	working_safety				: BOOL;
	baffle_sensor_1				: BOOL;
	baffle_sensor_2				: BOOL;
	
	LiftStoEDM					: BOOL;
	Place1StoEDM				: BOOL;
	Place2StoEDM				: BOOL;  

	
	safety_door_unlock_en		: BOOL;
	bStop_button_unlock		: BOOL;//for not receive cmd from tote_subsystem
	

	
	
	refMachineCmd	: REFERENCE TO E_PMLCommand;
	lift_safetyDoor_left: BOOL;
	lift_safetyDoor_right: BOOL;
	

	
	ton_waitDoorLocked	: TON;
	
	pml_command	: E_PMLCommand;
	
	bDoorUnlockRequest	: BOOL;
	fTrig_error	:ARRAY[1..20] OF F_TRIG;
	
	resetting	: BOOL;//while in resetting,can not unlock the door
	
END_VAR

SUPER^();
M_mapping();
M_safetyDoor();


IF sInstanceName='safety_1' THEN
	IF pMachine^.eState=ePMLState_Aborted AND xEstop AND pSafety_door^.door_locked AND 
	 	(GVL.fb_mcp_2.st_safety_door.door_locked OR lift_door_right.Q)
	THEN
		pSafety_door^.lamp_reset	:= GPWM_1s.q_xOut;
	ELSE
		pSafety_door^.lamp_reset	:= FALSE;
	END_IF	
END_IF
IF sInstanceName='safety_2' THEN
	IF pMachine^.eState=ePMLState_Aborted AND xEstop AND pSafety_door^.door_locked AND 
	 	(GVL.fb_mcp_1.st_safety_door.door_locked OR lift_door_left.Q)
	THEN
		pSafety_door^.lamp_reset	:= GPWM_1s.q_xOut;
	ELSE
		pSafety_door^.lamp_reset	:= FALSE;
	END_IF	
END_IF

xEstop	:= bRobot1_eStop AND bRobot2_eStop AND mcp_estop_left.Q AND mcp_estop_right.Q AND lift_station_detection AND baffle_sensor_1 AND baffle_sensor_2;
xEstop_behavior	:= NOT(GVL_SAFETY.robot1_STO_EES AND GVL_SAFETY.robot2_STO_EES AND GVL_SAFETY.Lift_STO);
IF sInstanceName='safety_1' THEN
		xError	:=NOT(GVL_SAFETY.robot1_STO_EES AND GVL_SAFETY.Lift_STO AND GVL_SAFETY.Place1_STO AND GVL_SAFETY.robot1_STO_EAS); 
		GVL_SAFETY.bLeftDoorUnlock_Request	:= pSafety_door^.door_lock;		
		IF robot1_EES THEN 
			IF robot1_EAS THEN
				safety_status := GeneralStatus.READY ;
			ELSE
				safety_status := GeneralStatus.NOT_READY ;
			END_IF
		ELSE
			safety_status := GeneralStatus.ERROR; 
		END_IF
END_IF
IF sInstanceName='safety_2' THEN
	xError	:=NOT(GVL_SAFETY.robot2_STO_EES AND GVL_SAFETY.Lift_STO AND GVL_SAFETY.Place2_STO AND GVL_SAFETY.robot2_STO_EAS);
	GVL_SAFETY.bRightDoorUnlock_Request	:= pSafety_door^.door_lock;
	IF robot2_EES THEN 
		IF robot2_EAS THEN
			safety_status := GeneralStatus.READY ;
		ELSE
			safety_status := GeneralStatus.NOT_READY ;
		END_IF
	ELSE
		safety_status := GeneralStatus.ERROR; 
	END_IF		
END_IF

//安全Safety报警 确认 复位
tonSaftyDelay(IN:= NOT tonSaftyDelay.Q ,PT:=T#1S);
b_ErrorAck := tonSaftyDelay.Q;


GPWM(i_xEnable:=TRUE,i_udiTime:=10,i_udiCycle:=20);
GPWM_1s(i_xEnable:=TRUE,i_udiTime:=500,i_udiCycle:=1000);

 



////////////////////////////////////////////////safety error/////////////////////////////////////////////////// 
IF wcState_mcp=0 AND wcState_lift=0 AND wcState_place1=0 AND wcState_place2=0 THEN
	fTrig_error[1](CLK:=mcp_estop_left.Q OR pMachine^.eState = ePMLState_Clearing);
	fTrig_error[2](CLK:=mcp_estop_right.Q OR pMachine^.eState = ePMLState_Clearing);
	fTrig_error[3](CLK:=bRobot1_eStop OR pMachine^.eState = ePMLState_Clearing);
	fTrig_error[4](CLK:=bRobot2_eStop OR pMachine^.eState = ePMLState_Clearing);
	fTrig_error[5](CLK:=lift_station_detection OR pMachine^.eState = ePMLState_Clearing);
	fTrig_error[6](CLK:=baffle_sensor_1 OR pMachine^.eState = ePMLState_Clearing);
	fTrig_error[7](CLK:= baffle_sensor_2 OR pMachine^.eState = ePMLState_Clearing);
	IF sInstanceName='safety_1' THEN
		fTrig_error[8](CLK:=safetyDoor_left OR pMachine^.eState = ePMLState_Clearing);
	END_IF
	IF sInstanceName='safety_2' THEN
		fTrig_error[8](CLK:=safetyDoor_right OR pMachine^.eState = ePMLState_Clearing);
	END_IF
END_IF
fTrig_error[9](CLK:= wcState_mcp=0 OR pMachine^.eState = ePMLState_Clearing);
fTrig_error[10](CLK:= wcState_lift=0 OR pMachine^.eState = ePMLState_Clearing);
fTrig_error[11](CLK:= wcState_place1=0 OR pMachine^.eState = ePMLState_Clearing);
fTrig_error[12](CLK:= wcState_place2=0 OR pMachine^.eState = ePMLState_Clearing);
IF pPackTags^.Status.StateCurrent<>E_PMLState.ePMLState_Resetting THEN
	FOR i:=1 TO 20 DO
		IF fTrig_error[i].Q THEN
			THIS^.packTags.Admin.Alarm[i].ID	:= i;
			CASE i OF
				1:
					THIS^.packTags.Admin.Alarm[1].Message	:= GenerateErrorMsg(errorType:='S',iState := i,errorMsg:='estop on left door is pressed');
				2:
					THIS^.packTags.Admin.Alarm[2].Message	:= GenerateErrorMsg(errorType:='S',iState := i,errorMsg:='estop on right door is pressed');
				3:
					THIS^.packTags.Admin.Alarm[3].Message	:= GenerateErrorMsg(errorType:='S',iState := i,errorMsg:='estop on robot1 teachpannel is pressed');
				4:
					THIS^.packTags.Admin.Alarm[4].Message	:= GenerateErrorMsg(errorType:='S',iState := i,errorMsg:='estop on robot2 teachpannel is pressed');
				5:
					THIS^.packTags.Admin.Alarm[5].Message	:= GenerateErrorMsg(errorType:='S',iState := i,errorMsg:='switch detecting lift module is not detected');
				6:
					THIS^.packTags.Admin.Alarm[6].Message	:= GenerateErrorMsg(errorType:='S',iState := i,errorMsg:='up baffle is not detected');	
				7:
					THIS^.packTags.Admin.Alarm[7].Message	:= GenerateErrorMsg(errorType:='S',iState := i,errorMsg:='down baffle is not detected');	
				8:
					THIS^.packTags.Admin.Alarm[8].Message	:= GenerateErrorMsg(errorType:='S',iState := i,errorMsg:='gate is unlocked');	
				9:
					THIS^.packTags.Admin.Alarm[9].Message	:= GenerateErrorMsg(errorType:='S',iState := i,errorMsg:='MCP EtherCAT bus is in state ERROR');	
				10:
					THIS^.packTags.Admin.Alarm[10].Message	:= GenerateErrorMsg(errorType:='S',iState := i,errorMsg:='Lift module EtherCAT bus is in state ERROR');	
				11:
					THIS^.packTags.Admin.Alarm[11].Message	:= GenerateErrorMsg(errorType:='S',iState := i,errorMsg:='Place1 module EtherCAT bus is in state ERROR');	
				12:
					THIS^.packTags.Admin.Alarm[12].Message	:= GenerateErrorMsg(errorType:='S',iState := i,errorMsg:='Place2 module EtherCAT bus is in state ERROR');	

			END_CASE
			THIS^.pml_adminAlarm.M_SetAlarm(stAdmin:=pPackTags^.Admin,stAlarm := THIS^.packTags.Admin.Alarm[i]);
		END_IF
	END_FOR
END_IF

PROPERTY _stationMode : StationMode
GET
_stationMode	:= station_mode;
END_GET
SET
station_mode	:= _stationMode;
END_SET
END_PROPERTY

METHOD M_mapping : BOOL
VAR_INPUT
END_VAR

VAR

	
END_VAR


mcp_estop_left(D:= G_IO.arSI[0].Ch[1] AND G_IO.arSI[0].Ch[2],on_ms:=100,off_ms:=50);//while trig door lock and unlock,it will trig the input randomly	
safetyDoor_left				:= G_IO.arSI[0].Ch[3] AND G_IO.arSI[0].Ch[4];
mcp_estop_right(D:= G_IO.arSI[1].Ch[1] AND G_IO.arSI[1].Ch[2],on_ms:=100,off_ms:=50);//while trig door lock and unlock,it will trig the input randomly	
safetyDoor_right			:= G_IO.arSI[1].Ch[3] AND G_IO.arSI[1].Ch[4];
IF sInstanceName='safety_1' THEN
	door_closed					:= G_IO.arSI[2].Ch[3];
END_IF
IF sInstanceName='safety_2' THEN
	door_closed					:= G_IO.arSI[2].Ch[4];
END_IF
bRobot1_eStop				:= G_IO.arSI[3].Ch[1] AND G_IO.arSI[3].Ch[2];
bRobot2_eStop				:= G_IO.arSI[3].Ch[3] AND G_IO.arSI[3].Ch[4];

lift_station_detection		:= G_IO.arSI[4].Ch[3] AND G_IO.arSI[4].Ch[4];
lift_door_left(D:= G_IO.arSI[5].Ch[1] AND G_IO.arSI[5].Ch[2],on_ms:=500,off_ms:=80);
lift_door_right(D:= G_IO.arSI[5].Ch[3] AND G_IO.arSI[5].Ch[4],on_ms:=500,off_ms:=80);
baffle_sensor_1				:= G_IO.arSI[6].Ch[1] AND G_IO.arSI[6].Ch[2];
baffle_sensor_2				:= G_IO.arSI[6].Ch[3] AND G_IO.arSI[6].Ch[4];
	
robot1_EES					:= GVL_SAFETY.robot1_STO_EES;
robot1_EAS					:= GVL_SAFETY.robot1_STO_EAS;
robot2_EES					:= GVL_SAFETY.robot2_STO_EES;
robot2_EAS					:= GVL_SAFETY.robot2_STO_EAS;
LiftStoEDM					:= GVL_SAFETY.Lift_STO_EDM;
Place1StoEDM				:= GVL_SAFETY.Place1_STO_EDM;
Place2StoEDM				:= GVL_SAFETY.Place2_STO_EDM;                 
                    
                  
 //EDM config
// GVL_IOLink.robots_ees_edm  	:= TRUE;  
 GVL_SAFETY.Robot1_EES_EDM  	:= GVL.fb_mcp_1.EDM_EES;
 GVL_SAFETY.Robot2_EES_EDM  	:= GVL.fb_mcp_2.EDM_EES; 
 GVL_SAFETY.robot1_eas_edm  	:= GVL.fb_mcp_1.EDM_EAS;
 GVL_SAFETY.robot2_eas_edm  	:= GVL.fb_mcp_2.EDM_EAS;
// GVL_SAFETY.Lift_STO_EDM        := GVL.fb_loading.EDM_KM;
// GVL_SAFETY.Place1_STO_EDM      := GVL.fb_working1.EDM_KM;
// GVL_SAFETY.Place2_STO_EDM      := GVL.fb_working2.EDM_KM;	
	



/////////////////////////////////////////////Estop array//////////////////////////////////
IF mcp_estop_left.Q THEN
	estop_array[0]:=EStopStatus.DISENGAGED;
ELSE
	estop_array[0]:=EStopStatus.ENGAGED;	
END_IF
IF mcp_estop_right.Q THEN
	estop_array[1]:=EStopStatus.DISENGAGED;
ELSE
	estop_array[1]:=EStopStatus.ENGAGED;	
END_IF
IF bRobot1_eStop THEN
	estop_array[2]:=EStopStatus.DISENGAGED;
ELSE
	estop_array[2]:=EStopStatus.ENGAGED;	
END_IF
IF bRobot2_eStop THEN
	estop_array[3]:=EStopStatus.DISENGAGED;
ELSE
	estop_array[3]:=EStopStatus.ENGAGED;	
END_IF

/////////////////////////////////////////////button array//////////////////////////////////

IF pSafety_door^.button_reset THEN
	button_array[0]:=ButtonStatus.PRESSED;
ELSE
	button_array[0]:=ButtonStatus.RELEASED;	
END_IF
IF pSafety_door^.button_unlock THEN
	button_array[1]:=ButtonStatus.PRESSED;
ELSE
	button_array[1]:=ButtonStatus.RELEASED;	
END_IF
/////////////////////////////////////////////safety door array//////////////////////////////////
IF sInstanceName='safety_1' THEN
	IF safetyDoor_left THEN
		safety_door_array[0]:=SafetyDoorStatus.LOCKED;
	ELSE
		safety_door_array[0]:=SafetyDoorStatus.UNLOCKED;
	END_IF
END_IF
IF sInstanceName='safety_2' THEN
	IF safetyDoor_right THEN
		safety_door_array[0]:=SafetyDoorStatus.LOCKED;
	ELSE
		safety_door_array[0]:=SafetyDoorStatus.UNLOCKED;
	END_IF	
END_IF   
/////////////////////////////////////////////sensor array//////////////////////////////////
IF lift_station_detection THEN
	sensor_array[0]:=SensorStatus.SIGNAL;
ELSE
	sensor_array[0]:=SensorStatus.NO_SIGNAL;
END_IF
IF baffle_sensor_1 THEN
	sensor_array[1]:=SensorStatus.SIGNAL;
ELSE
	sensor_array[1]:=SensorStatus.NO_SIGNAL;
END_IF
IF baffle_sensor_2 THEN
	sensor_array[2]:=SensorStatus.SIGNAL;
ELSE
	sensor_array[2]:=SensorStatus.NO_SIGNAL;
END_IF
IF lift_door_left.Q THEN
	sensor_array[3]:=SensorStatus.SIGNAL;
ELSE
	sensor_array[3]:=SensorStatus.NO_SIGNAL;
END_IF

IF lift_door_right.Q THEN
	sensor_array[4]:=SensorStatus.SIGNAL;
ELSE
	sensor_array[4]:=SensorStatus.NO_SIGNAL;
END_IF
IF pSafety_door^.door_closed THEN
	sensor_array[5]:=SensorStatus.SIGNAL;
ELSE
	sensor_array[5]:=SensorStatus.NO_SIGNAL;
END_IF
//GI_0.0	:= GVL.fb_mcp.st_safety_door.button_reset;
//GI_0.1	:= GVL.fb_mcp.st_safety_door.button_unlock;
//GI_0.2	:= GVL.fb_mcp.st_safety_door.door_closed;

//SI_0.0	:= mcp_estop_left;
//SI_0.1	:= safetyDoor_left;
//SI_0.2	:= belt_estop;
//SI_0.3	:= lift_estop;
//SI_0.4	:= lift_station_detection;
END_METHOD

METHOD M_reset : BOOL
VAR_INPUT
	
END_VAR
M_reset	:= FALSE;
resetting	:= TRUE;
//xError	:= FALSE;//remove while safety is ready
//M_reset	:= TRUE;//remove while safety is ready
//RETURN;//remove while safety is ready
//check if all safety outputs
//////////////////////////////////////////////////////////timeout//////////////////////////////////////////
		ton_timeout();
		iStateTemp	:= eStateTemp;
		IF eStateTemp=eStates THEN
			ton_timeout.IN	:=TRUE;
		ELSE
			ton_timeout.IN	:=FALSE;
			eStateTemp	:= eStates;	
			M_Log(eLogType:=ServerityLevelType.INFO,sTextLog:='');
			IF ton_timeout.Q THEN
				RETURN;
			END_IF
		END_IF
		IF ton_timeout.Q THEN	
			ton_timeout.IN	:=FALSE;
			CASE eStates OF	
				E_SafetyStates.ERROR:	
					alarm_temp.Message	:= GenerateErrorMsg(errorType:='S',iState := iStateTemp,errorMsg:='in error state.');
				ELSE
					alarm_temp.Message	:= GenerateErrorMsg(errorType:='S',iState := iStateTemp,errorMsg:='time out');
			END_CASE
//////////////////////////////////////////////////////////states don't want to timeout and trig error//////////////////////////////////////////				
			IF  eStates<>E_SafetyStates.IDLE AND
				eStates<>E_SafetyStates.TRIG_RESET
			THEN
				eStates	:= E_SafetyStates.ERROR;
				IF sInstanceName='safety_1' THEN					
					THIS^.pml_adminAlarm.M_SetAlarm(stAdmin:=GVL.PackTags1.Admin,stAlarm:=THIS^.alarm_temp);
				END_IF			
				IF sInstanceName='safety_2' THEN
					THIS^.pml_adminAlarm.M_SetAlarm(stAdmin:=GVL.PackTags2.Admin,stAlarm:=THIS^.alarm_temp);
				END_IF					
			END_IF
		END_IF


CASE eStates OF
	E_SafetyStates.IDLE:
		pml_command	:= ePMLCommand_Undefined;
		xError	:= FALSE;
		ton_timeout.PT	:= T#1000MS;
		eStates	:= E_SafetyStates.CHECK_SAFETY_INPUTS;
	E_SafetyStates.CHECK_SAFETY_INPUTS:
		IF xEstop AND pSafety_door^.door_locked THEN
			eStates	:= E_SafetyStates.CHECK_OTHER_STATION;
		END_IF
	E_SafetyStates.CHECK_OTHER_STATION:
		IF sInstanceName='safety_1' THEN
			IF GVL.fb_mcp_2.st_safety_door.door_locked OR lift_door_right.Q THEN
				eStates	:= E_SafetyStates.TRIG_RESET;
			END_IF
		END_IF
		IF sInstanceName='safety_2' THEN
			IF GVL.fb_mcp_1.st_safety_door.door_locked OR lift_door_left.Q THEN
				eStates	:= E_SafetyStates.TRIG_RESET;
			END_IF
		END_IF
	E_SafetyStates.TRIG_RESET:
		ton_timeout.PT	:= T#300MS;
		b_EStopRestart	:= GPWM.q_xOut;
		IF sInstanceName='safety_1' THEN
			bSafetyRestart_left		:= GPWM.q_xOut;
		END_IF
		IF sInstanceName='safety_2' THEN	
			bSafetyRestart_right	:= GPWM.q_xOut;
		END_IF
		IF ton_timeout.Q THEN
			b_EStopRestart	:= FALSE;
			bSafetyRestart_left		:= FALSE;
			bSafetyRestart_right	:= FALSE;
			eStates	:= E_SafetyStates.CHECK_SAFETY_OUTPUT;
		END_IF
		
	E_SafetyStates.LOCKDOOR_REQUEST:
		ton_timeout.PT	:= T#3000MS;
		IF sInstanceName='safety_1' THEN
			IF GVL.fb_loading.M_LockRequest_1() THEN
				eStates	:= E_SafetyStates.DONE;
			END_IF			
		END_IF
		IF sInstanceName='safety_2' THEN
			IF GVL.fb_loading.M_LockRequest_2() THEN
				eStates	:= E_SafetyStates.DONE;
			END_IF			
		END_IF		
//		IF sInstanceName='safety_1' THEN
//			IF NOT (GVL.fb_loading.xLocking2 OR GVL.fb_loading.xUnlocking2) THEN
//				IF GVL.fb_loading.M_LockRequest(sInstanceName:=sInstanceName) THEN
//					eStates	:= E_SafetyStates.DONE;
//				END_IF					
//			END_IF
//		END_IF
//		IF sInstanceName='safety_2' THEN
//			IF NOT (GVL.fb_loading.xLocking1 OR GVL.fb_loading.xUnlocking1) THEN
//				IF GVL.fb_loading.M_LockRequest(sInstanceName:=sInstanceName) THEN
//					eStates	:= E_SafetyStates.DONE;
//				END_IF					
//			END_IF
//		END_IF	
		
	E_SafetyStates.CHECK_SAFETY_OUTPUT:	
		IF sInstanceName='safety_1' THEN
			IF Lift_STO AND Place1_STO THEN
				eStates	:= E_SafetyStates.LOCKDOOR_REQUEST;
			END_IF
		END_IF			
		IF sInstanceName='safety_2' THEN
			IF Lift_STO AND Place2_STO THEN
				eStates	:= E_SafetyStates.LOCKDOOR_REQUEST;		
			END_IF	
		END_IF
	E_SafetyStates.DONE:
		M_reset	:= TRUE;
		resetting	:= FALSE;
		eStates	:= E_SafetyStates.IDLE;
	E_SafetyStates.ERROR:	
		M_reset	:= TRUE;
		resetting	:= FALSE;
		xError	:= TRUE;
		eStates	:= E_SafetyStates.IDLE;

	
END_CASE
END_METHOD

(*
	button_lock:lock the gate and then control the related door of lift  
	button_unlock:	1)wait station stopped 
					2)control the related doors
					3)unlock the gate
	button_reset:	1)reset safety 
					2)control the related door of lift module
*)
METHOD M_safetyDoor : BOOL
VAR_INPUT
	
END_VAR

safety_door_unlock_en	:= (safety_status<>GeneralStatus.READY OR 
							(station_mode = StationMode.STOPPED OR 
							station_mode = StationMode.DISABLED OR
							station_mode = StationMode.INTERVENTION OR 
							pHeartBeat^.heart_timeout_Alarm)) AND
							(pMachine^.eState=ePMLState_Aborted OR 
							pMachine^.eState=ePMLState_Stopped OR	
							pMachine^.eState=ePMLState_Idle);

ton_waitDoorLocked(PT:=T#1000MS);
IF NOT xEstop THEN
	eStates_safetyDoor	:= E_SAFETYDOOR.UNLOCKING;	
END_IF			
CASE eStates_safetyDoor	OF
	E_SAFETYDOOR.IDLE:
		IF pSafety_door^.door_locked THEN
			eStates_safetyDoor	:= E_SAFETYDOOR.LOCKED;
		ELSE
			eStates_safetyDoor	:= E_SAFETYDOOR.UNLOCKED;
		END_IF
	E_SAFETYDOOR.LOCKED:
		pSafety_door^.lamp_lock	:=	FALSE;
		pSafety_door^.lamp_unlock	:= TRUE;//door lcoked,unlock lamp solid
		IF pSafety_door^.button_unlock AND NOT resetting THEN//while resetting,door can not be unlock,otherwise might trig safety
			bStop_button_unlock	:= TRUE;
			eStates_safetyDoor	:= E_SAFETYDOOR.WAIT_UNLOCK_EN;
		END_IF			
	E_SAFETYDOOR.REQUEST_LOCK:
	;
	E_SAFETYDOOR.SAFETY:
	;
	E_SAFETYDOOR.UNLOCKED:
		pSafety_door^.lamp_unlock	:= FALSE;
		IF pSafety_door^.door_closed THEN
			pSafety_door^.lamp_lock	:= GPWM_1s.q_xOut;//door closed,lock lamp blinking
			IF pSafety_door^.button_lock THEN
				bStop_button_unlock	:= FALSE;
				eStates_safetyDoor	:= E_SAFETYDOOR.WAIT_LOCKED;
			END_IF
		ELSE
			pSafety_door^.lamp_lock	:= TRUE;//door open,lock lamp solid
		END_IF
	E_SAFETYDOOR.WAIT_LOCKED:
		ton_waitDoorLocked.IN	:= TRUE;
		pSafety_door^.door_lock	:= FALSE;
		IF pSafety_door^.door_locked THEN
			ton_waitDoorLocked.IN	:= FALSE;
			eStates_safetyDoor	:= E_SAFETYDOOR.LOCKED;
	 	END_IF
		//if lock door failed,turn to unlock door and need to press the lock button to lock the door once more
		IF ton_waitDoorLocked.Q THEN
			ton_waitDoorLocked.IN	:= FALSE;
			eStates_safetyDoor	:= E_SAFETYDOOR.UNLOCKING;
		END_IF
		
	E_SAFETYDOOR.WATI_LODING_DOOR://wait the state of lift door
		pSafety_door^.lamp_unlock	:= GPWM_1s.q_xOut;//door unlocking,unlock lamp blinking
		IF sInstanceName='safety_1' THEN
			IF bAirDump1 THEN//while gate is locked and its air is dumpped,means safety error must be accupped 
				IF GVL.fb_loading.M_unlockRequest(sInstanceName:=sInstanceName) THEN
					eStates_safetyDoor	:= E_SAFETYDOOR.UNLOCKING;
				END_IF
			ELSE
				eStates_safetyDoor	:= E_SAFETYDOOR.UNLOCKING;	
			END_IF		
		END_IF	
		IF sInstanceName='safety_2' THEN
			IF bAirDump2 THEN//while gate is locked and its air is dumpped,means safety error must be accupped 
				IF GVL.fb_loading.M_unlockRequest(sInstanceName:=sInstanceName) THEN
					eStates_safetyDoor	:= E_SAFETYDOOR.UNLOCKING;
				END_IF
			ELSE
				eStates_safetyDoor	:= E_SAFETYDOOR.UNLOCKING;	
			END_IF			
		END_IF
	E_SAFETYDOOR.WAIT_UNLOCK_EN:
		IF pHeartBeat^.heart_timeout_Alarm OR (station_mode = StationMode.INTERVENTION AND pSafety_door^.button_unlock) THEN
			pml_command	:= ePMLCommand_Stop;
		END_IF
		
		pSafety_door^.lamp_unlock	:= GPWM_1s.q_xOut;//door unlocking,unlock lamp blinking
		IF safety_door_unlock_en THEN
			pml_command	:= ePMLCommand_Undefined;
			eStates_safetyDoor	:= E_SAFETYDOOR.WATI_LODING_DOOR;
		END_IF
	E_SAFETYDOOR.UNLOCKING:
		pml_command	:= ePMLCommand_Undefined;
		pSafety_door^.lamp_unlock	:= GPWM_1s.q_xOut;//door unlocking,unlock lamp blinking
		pSafety_door^.door_lock	:= TRUE;
		IF NOT pSafety_door^.door_locked THEN
			eStates_safetyDoor	:= E_SAFETYDOOR.UNLOCKED;
		END_IF
	
END_CASE
END_METHOD

METHOD ParseStateToString : STRING
VAR_INPUT
END_VAR
CASE THIS^.eStates OF
	E_SafetyStates.IDLE:
		ParseStateToString	:='IDLE';
	E_SafetyStates.CHECK_SAFETY_INPUTS:
		ParseStateToString	:='CHECK_SAFETY_INPUTS';
	E_SafetyStates.CHECK_DOOR_CLOSED:
		ParseStateToString	:='CHECK_DOOR_CLOSED';
	E_SafetyStates.CHECK_DOOR_LOCKED:
		ParseStateToString	:='CHECK_DOOR_LOCKED';
	E_SafetyStates.LOCKDOOR_REQUEST:
		ParseStateToString	:='LOCKDOOR_REQUEST';
	E_SafetyStates.CHECK_DOOR_OSSD:
		ParseStateToString	:='CHECK_DOOR_OSSD';
	E_SafetyStates.CHECK_SAFETY_OUTPUT:
		ParseStateToString	:='CHECK_SAFETY_OUTPUT';
	E_SafetyStates.DOOR_LOCK:
		ParseStateToString	:='DOOR_LOCK';
	E_SafetyStates.TRIG_RESET:
		ParseStateToString	:='TRIG_RESET';
	E_SafetyStates.CHECK_OTHER_STATION:
		ParseStateToString	:='CHECK_OTHER_STATION';
	E_SafetyStates.DONE:
		ParseStateToString	:='DONE';
	E_SafetyStates.ERROR:
		ParseStateToString	:='ERROR';
	ELSE
		ParseStateToString	:='UNKNOW STATE';
END_CASE
END_METHOD

{attribute 'TcRpcEnable'}
METHOD update_station_mode  : UDINT
VAR_INPUT
	update_station_mode_params	: UpdateStationModeParams;
END_VAR
update_station_mode	:= 1;
station_mode	:= update_station_mode_params.station_mode;
update_station_mode	:= 0;
END_METHOD

END_FUNCTION_BLOCK

// ---- Mian/FB_Machine.TcPOU
FUNCTION_BLOCK FB_Machine EXTENDS FB_Generic
VAR_INPUT
	pPML_Instance1	: POINTER TO FB_Generic;
	pPML_Instance2	: POINTER TO FB_Generic;//instance for couple and uncouple
	pPackTags		: POINTER TO ST_PackMLv30;
	pSafetySystem	: POINTER TO FB_Safety_Subsystem;
END_VAR
VAR_OUTPUT

END_VAR
VAR	
	stSubModuleInfo		: ARRAY [1..iSubModule] OF ST_PMLSubUnitInfo;	//Informations about the Subunits
//	pPML_Instance	: ARRAY [1..iSubModule] OF POINTER TO FB_Generic;
	arrCouple	: ARRAY [1..iSubModule] OF BOOL;
	arrCmd		: ARRAY [1..iSubModule] OF E_PMLCommand;
	unCouple	: BOOL;//all modules uncoupling
	
	rtrig_alarm	:ARRAY [1..iSubModule] OF ARRAY[1..MaxAlarms] OF R_TRIG;
	
	iCmd_unitsActive	: INT;
	iCmd_transfer	: INT;


	preEstate	: E_PMLState;
	
END_VAR
VAR CONSTANT
	iSubModule	: UINT :=2;
END_VAR

//pPML_Instance[1]	:= ADR(GVL.fb_sample1);
//pPML_Instance[2]	:= ADR(GVL.fb_sample2);
///////////////////////////////////////////for signal system/////////////////////////////////////////////////////////////
IF NOT unCouple THEN
	FOR i:=1 TO UINT_TO_INT(iSubModule) DO
		arrCmd[i]:=eCommand;
		arrCouple[i]:= TRUE;
//		pPML_Instance[i]^._bCouple	:= TRUE;

	END_FOR
END_IF
unCouple	:= TRUE;//for mix sysytem
//////////////////////////////////////////////couple cmd//////////////////////////////////////////////////////////
//FOR i:=1 TO UINT_TO_INT(iSubModule) DO
//	IF arrCouple[i] THEN
//		arrCmd[i]:=eCommand;
//	END_IF
//END_FOR

CASE iCmd_transfer OF	
	0:
		IF eCommand<>ePMLCommand_Undefined THEN
			iCmd_transfer	:= 1;
		END_IF
	1:	
		IF arrCouple[1] THEN
			arrCmd[1]	:= eCommand;
		END_IF
		IF arrCouple[2] THEN
			arrCmd[2]	:= eCommand;
		END_IF
		iCmd_transfer	:= 2;	
	2:
		CASE preEstate OF
			ePMLState_Undefined:
				IF eState=ePMLState_Aborted THEN
					iCmd_transfer	:= 3;
				END_IF			
			ePMLState_Aborted,ePMLState_Clearing:
				IF eState=ePMLState_Stopped OR eState=ePMLState_Aborted THEN
					iCmd_transfer	:= 3;
				END_IF
			ePMLState_Stopped,ePMLState_Resetting:
				IF eState=ePMLState_Idle OR eState=ePMLState_Aborted THEN
					iCmd_transfer	:= 3;
				END_IF				
			ePMLState_Idle,ePMLState_Starting:
				IF eState=ePMLState_Execute OR eState=ePMLState_Stopped OR eState=ePMLState_Aborted THEN
					iCmd_transfer	:= 3;
				END_IF				
			ePMLState_Execute,ePMLState_Aborting,ePMLState_Stopping:
				IF eState=ePMLState_Stopped OR eState=ePMLState_Aborted THEN
					iCmd_transfer	:= 3;
				END_IF				
		END_CASE	
	3:
		arrCouple[2]	:= FALSE;
		arrCmd[1]	:=	ePMLCommand_Undefined;
		arrCmd[2]	:=	ePMLCommand_Undefined;
		iCmd_transfer	:= 0;	
END_CASE



pPML_Instance1^(
	eModeCommand:= eModeCommand, 
	eCommand:= arrCmd[1], 
	eMode=> , 
	eState=> stSubModuleInfo[1].eState, 
	bUndefinedDone=> , 
	bInvalidModeCommandOut=> , 
	bChangeIntoProduction=> );
stSubModuleInfo[1].Active		:= arrCouple[1];

pPML_Instance2^(
	eModeCommand:= eModeCommand, 
	eCommand:= , 
	eMode=> , 
	eState=> stSubModuleInfo[2].eState, 
	bUndefinedDone=> , 
	bInvalidModeCommandOut=> , 
	bChangeIntoProduction=> );
IF stSubModuleInfo[2].Active THEN
	pPML_Instance2^.eCommand	:= arrCmd[2];
END_IF	
stSubModuleInfo[2].Active		:= arrCouple[2];


IF  pPML_Instance1^.bUndefinedDone AND 
	pPML_Instance2^.bUndefinedDone 
THEN
	bUndefinedDone := TRUE;
END_IF

//The fbStateMachine from FB_Machine gets the Information about the states and activity from the subunits
fbStateMachine.stSubUnitInfoRef.ArraySize		:= SIZEOF(stSubModuleInfo);
fbStateMachine.stSubUnitInfoRef.NoOfSubUnits	:= iSubModule;
fbStateMachine.stSubUnitInfoRef.pArray			:= ADR(stSubModuleInfo);



//Set unit information 
M_SetUnitInfo();






SUPER^();

{attribute 'object_name' := 'M_Clearing'}
METHOD M_Clearing

CASE fbUnitModeManager.eModeStatus OF
	ePMLProtUnitMode_Production:		//Production, Mantainance, Manual
		FOR i:=1 TO 3 DO//try clear alarm several times
			FOR j:=1 TO MaxAlarms DO
				GVL.pml_adminAlarm.M_AcknowledgeAlarm(stAdmin:=pPackTags^.Admin,stAlarm:=pPackTags^.Admin.Alarm[j]);
				GVL.pml_adminAlarm.M_ClearAlarm(stAdmin:=pPackTags^.Admin,stAlarm:=pPackTags^.Admin.Alarm[j]);
			END_FOR	
		END_FOR	
		IF pSafetySystem^.M_reset() THEN
			IF pSafetySystem^.xError THEN
				IF M_UnitsActive(ePMLCommand_Abort)THEN
					eCommand	:= ePMLCommand_Abort;
				END_IF
			ELSE
				M_StateComplete();
			END_IF
		END_IF	
		
	
	ePMLProtUnitMode_Maintenance, ePMLProtUnitMode_Manual, ePMLUnitMode_Service:
		M_StateComplete();
END_CASE
END_METHOD

{attribute 'object_name' := 'M_Execute'}
METHOD M_Execute
END_METHOD

{attribute 'object_name' := 'M_Resetting'}
METHOD M_Resetting
CASE fbUnitModeManager.eModeStatus OF
	ePMLProtUnitMode_Production:		//Production, Mantainance, Manual	
		IF pSafetySystem^.M_reset() THEN
			IF pSafetySystem^.xError THEN
				IF M_UnitsActive(ePMLCommand_Abort)THEN
					eCommand	:= ePMLCommand_Abort;
				END_IF
			ELSE
				M_StateComplete();
			END_IF
		END_IF	
		
	
	ePMLProtUnitMode_Maintenance, ePMLProtUnitMode_Manual, ePMLUnitMode_Service:
		M_StateComplete();
END_CASE
END_METHOD

METHOD M_SetUnitInfo
VAR_INPUT
END_VAR
GVL.aUnitInfo[eMachine].Name			:= 'fbMachine';
GVL.aUnitInfo[eMachine].ActMode			:= eMode;
GVL.aUnitInfo[eMachine].ActState		:= eState;

GVL.aUnitInfo[eWorking1].Name			:= GVL.fb_working1._sInstanceName;
GVL.aUnitInfo[eWorking1].ActMode		:= GVL.fb_working1.eMode;
GVL.aUnitInfo[eWorking1].ActState		:= GVL.fb_working1.eState;

GVL.aUnitInfo[eLoading].Name			:= GVL.fb_loading._sInstanceName;
GVL.aUnitInfo[eLoading].ActMode			:= GVL.fb_loading.eMode;
GVL.aUnitInfo[eLoading].ActState		:= GVL.fb_loading.eState;

GVL.aUnitInfo[eWorking2].Name			:= GVL.fb_working2._sInstanceName;
GVL.aUnitInfo[eWorking2].ActMode		:= GVL.fb_working2.eMode;
GVL.aUnitInfo[eWorking2].ActState		:= GVL.fb_working2.eState;
END_METHOD

{attribute 'object_name' := 'M_Starting'}
METHOD M_Starting
CASE fbUnitModeManager.eModeStatus OF
	ePMLProtUnitMode_Production:		//Production, Mantainance, Manual
		//Resetting all Commands and Value
		G_HMI.bAging_test	:= FALSE;
		M_StateComplete();
	ePMLProtUnitMode_Maintenance, ePMLProtUnitMode_Manual, ePMLUnitMode_Service:
		M_StateComplete();
END_CASE
END_METHOD

//nomal
//idle/excute->stop 	idle/excute->abort
//loding error->abort
METHOD M_UnitsActive : BOOL
VAR_INPUT
	preCmd	: E_PMLCommand;
END_VAR
VAR 
	
END_VAR
M_UnitsActive	:= FALSE;




CASE iCmd_unitsActive OF
	0:
		iCmd_unitsActive	:= 1;
		iCmd_transfer	:= 0;
//get the command from main
	1:
		iCmd_unitsActive	:= 2;
//verify state
	2:
		IF NOT pSafetySystem^.xEstop THEN//no matter in which state,couple all the units
			arrCouple[1]	:= TRUE;
			arrCouple[2]	:= TRUE;	
			iCmd_unitsActive	:= 4;		
		ELSE
			IF (stSubModuleInfo[1].eState=ePMLState_Aborted OR stSubModuleInfo[1].eState=ePMLState_Stopped OR
				stSubModuleInfo[1].eState=ePMLState_Idle OR stSubModuleInfo[1].eState=ePMLState_Execute) AND
				(stSubModuleInfo[2].eState=ePMLState_Aborted OR stSubModuleInfo[2].eState=ePMLState_Stopped OR
				stSubModuleInfo[2].eState=ePMLState_Idle OR stSubModuleInfo[2].eState=ePMLState_Execute) AND
				(eState=ePMLState_Aborted OR eState=ePMLState_Stopped OR eState=ePMLState_Idle OR eState=ePMLState_Execute)
			THEN
				iCmd_unitsActive	:= 3;
			END_IF
		END_IF
//determine if couple or not
	3:
		CASE stSubModuleInfo[1].eState OF
			ePMLState_Aborted:
				CASE stSubModuleInfo[2].eState OF
					ePMLState_Aborted:
						CASE preCmd OF
							ePMLCommand_Clear:
								arrCouple[1]	:= TRUE;
								arrCouple[2]	:= TRUE;	
							ePMLCommand_Reset:	
								//					
							ePMLCommand_Start:	
								//
							ePMLCommand_Stop:	
								//
							ePMLCommand_Abort:
								IF pPML_Instance2^.isError OR pSafetySystem^.xEstop_behavior THEN
									arrCouple[2]	:= TRUE;
								ELSE
									arrCouple[2]	:= FALSE;
								END_IF									
						END_CASE						
					ePMLState_Stopped:
						CASE preCmd OF
							ePMLCommand_Clear:
								arrCouple[1]	:= TRUE;
								arrCouple[2]	:= FALSE;	
							ePMLCommand_Reset:	
								//					
							ePMLCommand_Start:	
								//
							ePMLCommand_Stop:	
								//
							ePMLCommand_Abort:
								IF pPML_Instance2^.isError OR pSafetySystem^.xEstop_behavior THEN
									arrCouple[2]	:= TRUE;
								ELSE
									arrCouple[2]	:= FALSE;
								END_IF									
						END_CASE					
					ePMLState_Idle:
						CASE preCmd OF
							ePMLCommand_Clear:
								arrCouple[1]	:= TRUE;
								arrCouple[2]	:= FALSE;	
							ePMLCommand_Reset:	
								//					
							ePMLCommand_Start:	
								//
							ePMLCommand_Stop:	
								//
							ePMLCommand_Abort:
								IF pPML_Instance2^.isError OR pSafetySystem^.xEstop_behavior THEN
									arrCouple[2]	:= TRUE;
								ELSE
									arrCouple[2]	:= FALSE;
								END_IF									
						END_CASE
					ePMLState_Execute:
						CASE preCmd OF
							ePMLCommand_Clear:
								arrCouple[1]	:= TRUE;
								arrCouple[2]	:= FALSE;	
							ePMLCommand_Reset:	
								//					
							ePMLCommand_Start:	
								//
							ePMLCommand_Stop:	
								//
							ePMLCommand_Abort:
								IF pPML_Instance2^.isError OR pSafetySystem^.xEstop_behavior THEN
									arrCouple[2]	:= TRUE;
								ELSE
									arrCouple[2]	:= FALSE;
								END_IF									
						END_CASE	
				END_CASE		
			ePMLState_Stopped:
				CASE stSubModuleInfo[2].eState OF	
					ePMLState_Aborted:
						//
					ePMLState_Stopped:
						CASE preCmd OF
							ePMLCommand_Clear:
								//
							ePMLCommand_Reset:	
								arrCouple[1]	:= TRUE;
								arrCouple[2]	:= TRUE;						
							ePMLCommand_Start:	
								//
							ePMLCommand_Stop:	
								//
							ePMLCommand_Abort:
								IF pPML_Instance2^.isError OR pSafetySystem^.xEstop_behavior THEN
									arrCouple[2]	:= TRUE;
								ELSE
									arrCouple[2]	:= FALSE;
								END_IF									
						END_CASE					
					ePMLState_Idle:
						CASE preCmd OF
							ePMLCommand_Clear:
								//
							ePMLCommand_Reset:	
								arrCouple[1]	:= TRUE;
								arrCouple[2]	:= FALSE;						
							ePMLCommand_Start:	
								//
							ePMLCommand_Stop:	
								//
							ePMLCommand_Abort:
								IF pPML_Instance2^.isError OR pSafetySystem^.xEstop_behavior THEN
									arrCouple[2]	:= TRUE;
								ELSE
									arrCouple[2]	:= FALSE;
								END_IF									
						END_CASE					
					ePMLState_Execute:
						CASE preCmd OF
							ePMLCommand_Clear:
								//
							ePMLCommand_Reset:	
								arrCouple[1]	:= TRUE;
								arrCouple[2]	:= FALSE;						
							ePMLCommand_Start:	
								//
							ePMLCommand_Stop:	
								//
							ePMLCommand_Abort:
								IF pPML_Instance2^.isError OR pSafetySystem^.xEstop_behavior THEN
									arrCouple[2]	:= TRUE;
								ELSE
									arrCouple[2]	:= FALSE;
								END_IF									
						END_CASE					
				END_CASE	

	
			ePMLState_Idle:
				CASE stSubModuleInfo[2].eState OF	
					ePMLState_Aborted:
						//
					ePMLState_Stopped:
						//
					ePMLState_Idle:
						CASE preCmd OF
							ePMLCommand_Clear:
								//
							ePMLCommand_Reset:	
								//						
							ePMLCommand_Start:	
								arrCouple[1]	:= TRUE;
								arrCouple[2]	:= TRUE;
							ePMLCommand_Stop:	
								arrCouple[1]	:= TRUE;
								arrCouple[2]	:= FALSE;									
							ePMLCommand_Abort:
								IF pPML_Instance2^.isError OR pSafetySystem^.xEstop_behavior THEN
									arrCouple[2]	:= TRUE;
								ELSE
									arrCouple[2]	:= FALSE;
								END_IF									
						END_CASE					
					ePMLState_Execute:
						CASE preCmd OF
							ePMLCommand_Clear:
								//
							ePMLCommand_Reset:	
								//						
							ePMLCommand_Start:	
								arrCouple[1]	:= TRUE;
								arrCouple[2]	:= FALSE;
							ePMLCommand_Stop:	
								arrCouple[1]	:= TRUE;
								arrCouple[2]	:= FALSE;									
							ePMLCommand_Abort:
								IF pPML_Instance2^.isError OR pSafetySystem^.xEstop_behavior THEN
									arrCouple[2]	:= TRUE;
								ELSE
									arrCouple[2]	:= FALSE;
								END_IF									
						END_CASE
				END_CASE	
			ePMLState_Execute:
				CASE stSubModuleInfo[2].eState OF	
					ePMLState_Aborted:
						//
					ePMLState_Stopped:
						//
					ePMLState_Idle:
						//
					ePMLState_Execute:
						CASE preCmd OF
							ePMLCommand_Clear:
								//
							ePMLCommand_Reset:	
								//						
							ePMLCommand_Start:	
								//
							ePMLCommand_Stop:	
								arrCouple[1]	:= TRUE;
								arrCouple[2]	:= FALSE;									
							ePMLCommand_Abort:
								IF pPML_Instance2^.isError OR pSafetySystem^.xEstop_behavior THEN
									arrCouple[2]	:= TRUE;
								ELSE
									arrCouple[2]	:= FALSE;
								END_IF									
						END_CASE	
				END_CASE	
		END_CASE
		iCmd_unitsActive	:= 4;
		
	4:
		preEstate	:= eState;
		iCmd_unitsActive	:= 0;
		M_UnitsActive	:= TRUE	;
	
//set the command to units
END_CASE
END_METHOD

END_FUNCTION_BLOCK

// ---- Ads/FB_Tote_Subsystem.TcPOU
FUNCTION_BLOCK FB_Tote_Subsystem EXTENDS FB_Generic
VAR_INPUT
	
END_VAR
VAR_OUTPUT
END_VAR
VAR
	tote_status_array 	AT%Q*	: ARRAY [0..99] OF ToteStatus;
	
	status					: MachineStatus := MachineStatus.STOPPED;	
	current_air_pressure	: REAL;	
	machine_control_cmd	 	: MachineControlCommand;
	
	cmd						: OrderToteCommand;
	
	ton1					: TON;

	ton_heart_beat			: TON;
	bReset_ads_heart_beat	: BOOL;
	bTest					: BOOL;
	
	machine_current_status	: E_PMLState;
	workflow1_status		: ToteSubsystemWorkflowStatus := ToteSubsystemWorkflowStatus.UNKNOWN;
	error1_status			: OrderToteErrorStatus := OrderToteErrorStatus.UNKNOWN;
	
	workflow2_status		: ToteSubsystemWorkflowStatus := ToteSubsystemWorkflowStatus.UNKNOWN;
	error2_status			: OrderToteErrorStatus := OrderToteErrorStatus.UNKNOWN;
	
	loading_tote			: ToteData;
	working1_tote			: ToteData;
	working2_tote			: ToteData;
	
	
	bInbound		: BOOL;
	bOutbound		: BOOL;
	bAbortInbound	: BOOL;
	bAbortOutbound	: BOOL;
	bAutostore_exchange	: BOOL;
	inboundToteParams_temp	: InboundToteParams;
	outboundToteParams_temp	: OutboundToteParams;
	abortToreParams_temp	: AbortToteRequestParams;

	A1	: INT;
	A2	: INT;
	iCase_abort	: INT;
END_VAR

SUPER^();
M_mapping();
IF sInstanceName='tote_1' THEN
	tote_status_array[0]	:= GVL.fb_loading.tote_status;
	tote_status_array[1]	:= GVL.fb_working1.tote_status;
	tote_status_array[2]	:= GVL.fb_working1.outboundTote_status;//outbound tote status form logtech
	machine_current_status	:= GVL.PackTags1.Status.StateCurrent;
END_IF
IF sInstanceName='tote_2' THEN
	tote_status_array[0]	:= GVL.fb_loading.tote_status;
	tote_status_array[1]	:= GVL.fb_working2.tote_status;
	tote_status_array[2]	:=  GVL.fb_working2.outboundTote_status;//outbound tote status form logtech
	machine_current_status	:= GVL.PackTags2.Status.StateCurrent;
END_IF

CASE machine_current_status OF
	ePMLState_Aborted,ePMLState_Aborting:
		status	:= MachineStatus.ERROR;
	ePMLState_Stopping:	
		status	:= MachineStatus.STOPPING;
	ePMLState_Stopped:
		status	:= MachineStatus.STOPPED;
	ePMLState_Resetting:	
		status	:= MachineStatus.RESETTING;
	ePMLState_Idle:	
		status	:= MachineStatus.READY;		
	ePMLState_Execute:	
		status	:= MachineStatus.RUNNING;			
END_CASE

IF bInbound THEN
	inboundToteParams_temp.source_id	:= ModelIdentifier.inbounding_position;
	inboundToteParams_temp.target_id	:= ModelIdentifier.working_position;
	inbound_tote_request(inbound_tote_params:=inboundToteParams_temp);
	bInbound	:= FALSE;
END_IF
IF bOutbound THEN
	outboundToteParams_temp.source_id	:= ModelIdentifier.working_position;
	outboundToteParams_temp.target_id	:= ModelIdentifier.outbound_position;	
	outbound_tote_request(outbound_tote_params:=outboundToteParams_temp);
	bOutbound	:= FALSE;
END_IF
IF bAbortInbound THEN
	abortToreParams_temp.source_id	:= ModelIdentifier.inbounding_position;
	abortToreParams_temp.target_id	:= ModelIdentifier.working_position;	
	abort_tote_request(abort_tote_request_params:=abortToreParams_temp);
	bAbortInbound	:= FALSE;
END_IF

IF bAbortOutbound THEN
	abortToreParams_temp.source_id	:= ModelIdentifier.working_position;
	abortToreParams_temp.target_id	:= ModelIdentifier.outbound_position;	
	abort_tote_request(abort_tote_request_params:=abortToreParams_temp);
	bAbortOutbound	:= FALSE;
END_IF
IF bAutostore_exchange THEN
	autostore_control_command(Command:=AutostoreControlCommand.START);
	bAutostore_exchange	:= FALSE;
END_IF

{attribute 'TcRpcEnable'}
METHOD abort_tote_request : UDINT//only response while awaiting
VAR_INPUT
	abort_tote_request_params : AbortToteRequestParams; // Struct containing data from the barcode scan	
END_VAR
abort_tote_request:=MethodCallReturnValue.DECLINED_BUSY;
IF sInstanceName='tote_1' THEN
	IF abort_tote_request_params.source_id=ModelIdentifier.inbounding_position AND abort_tote_request_params.target_id=ModelIdentifier.working_position THEN
		iCase_abort	:= 1;
	END_IF
	IF abort_tote_request_params.source_id=ModelIdentifier.working_position AND abort_tote_request_params.target_id=ModelIdentifier.outbound_position THEN
		iCase_abort	:= 2;
	END_IF		
	CASE iCase_abort OF
		1:
			IF GVL.fb_working1.tote_status=ToteStatus.AWAITING_INBOUND_AVAILABILITY THEN
				subData.Topic	:= E_Topics.WORKING1_ABORT_INBOUND;
				GVL.PubSubService.Publish(topic:=E_Topics.WORKING1_ABORT_INBOUND,data:= subData);
				abort_tote_request:= MethodCallReturnValue.ACCEPTED;
			ELSE
				abort_tote_request:= MethodCallReturnValue.DECLINED_ERROR;
			END_IF
		2:
			IF GVL.fb_working1.tote_status=ToteStatus.AWAITING_OUTBOUND_AVAILABILITY THEN
				subData.Topic	:= E_Topics.WORKING1_ABORT_OUTBOUND;
				GVL.PubSubService.Publish(topic:=E_Topics.WORKING1_ABORT_OUTBOUND,data:= subData);
				abort_tote_request:= MethodCallReturnValue.ACCEPTED;
			ELSE
				abort_tote_request:= MethodCallReturnValue.DECLINED_ERROR;
			END_IF	
		ELSE
			abort_tote_request:= MethodCallReturnValue.DECLINED_ERROR;
	END_CASE
END_IF

IF sInstanceName='tote_2' THEN
	IF abort_tote_request_params.source_id=ModelIdentifier.inbounding_position AND abort_tote_request_params.target_id=ModelIdentifier.working_position THEN
		iCase_abort	:= 1;
	END_IF
	IF abort_tote_request_params.source_id=ModelIdentifier.working_position AND abort_tote_request_params.target_id=ModelIdentifier.outbound_position THEN
		iCase_abort	:= 2;
	END_IF		
	CASE iCase_abort OF
		1:
			IF GVL.fb_working2.tote_status=ToteStatus.AWAITING_INBOUND_AVAILABILITY THEN
				subData.Topic	:= E_Topics.WORKING2_ABORT_INBOUND;
				GVL.PubSubService.Publish(topic:=E_Topics.WORKING2_ABORT_INBOUND,data:= subData);
				abort_tote_request:= MethodCallReturnValue.ACCEPTED;
			ELSE
				abort_tote_request:= MethodCallReturnValue.DECLINED_ERROR;
			END_IF
		2:
			IF GVL.fb_working2.tote_status=ToteStatus.AWAITING_INBOUND_AVAILABILITY THEN
				subData.Topic	:= E_Topics.WORKING2_ABORT_OUTBOUND;
				GVL.PubSubService.Publish(topic:=E_Topics.WORKING2_ABORT_OUTBOUND,data:= subData);
				abort_tote_request:= MethodCallReturnValue.ACCEPTED;
			ELSE
				abort_tote_request:= MethodCallReturnValue.DECLINED_ERROR;
			END_IF	
		ELSE
			abort_tote_request:= MethodCallReturnValue.DECLINED_ERROR;			
	END_CASE
END_IF
END_METHOD

{attribute 'TcRpcEnable'}
METHOD autostore_control_command : BOOL
VAR_INPUT
	Command	: AutostoreControlCommand;
END_VAR
IF sInstanceName='tote_1' THEN
	subData.Topic	:= E_Topics.AUTOSTORE1_EXCHANGE;
	GVL.PubSubService.Publish(topic:= E_Topics.AUTOSTORE1_EXCHANGE,data:= subData);
END_IF
IF sInstanceName='tote_2' THEN
	subData.Topic	:= E_Topics.AUTOSTORE2_EXCHANGE;
	GVL.PubSubService.Publish(topic:= E_Topics.AUTOSTORE2_EXCHANGE,data:= subData);
END_IF
END_METHOD

{attribute 'TcRpcEnable'}
METHOD barcode_validation_request : UDINT
VAR_INPUT
	barcode_validation_request_params : BarcodeValidationRequestParams;
END_VAR
END_METHOD

{attribute 'TcRpcEnable'}
METHOD inbound_tote_request : UDINT
VAR_INPUT
	inbound_tote_params : InboundToteParams;
END_VAR
VAR	
	subData	: PubSubData;
END_VAR

IF sInstanceName='tote_1' THEN
//	IF NOT (((GVL.fb_working1.xLoading OR GVL.fb_working1.xInbound) AND GVL.fb_loading.xOutbound_woking1) OR 
//		GVL.fb_working1.tote_status=ToteStatus.LOADED OR GVL.fb_working1.xUnloading OR GVL.fb_working1.xOutbound) 
//	THEN//avoid cmd while inbounding or has tote
//		subData.Topic	:= E_Topics.WORKING1_INBOUND_TOTE;
//		GVL.PubSubService.Publish(topic:= E_Topics.WORKING1_INBOUND_TOTE,data:= subData);	
//	END_IF
	subData.Topic	:= E_Topics.WORKING1_INBOUND_TOTE;
	GVL.PubSubService.Publish(topic:= E_Topics.WORKING1_INBOUND_TOTE,data:= subData);
	A1	:= A1+1;	
END_IF
IF sInstanceName='tote_2' THEN
//	IF NOT (((GVL.fb_working2.xLoading OR GVL.fb_working2.xInbound) AND GVL.fb_loading.xOutbound_woking2) OR 
//		GVL.fb_working2.tote_status=ToteStatus.LOADED OR GVL.fb_working2.xUnloading OR GVL.fb_working2.xOutbound) 
//	THEN//avoid cmd while inbounding or has tote
//		subData.Topic	:= E_Topics.WORKING2_INBOUND_TOTE;
//		GVL.PubSubService.Publish(topic:= E_Topics.WORKING2_INBOUND_TOTE,data:= subData);
//	END_IF
	subData.Topic	:= E_Topics.WORKING2_INBOUND_TOTE;
	GVL.PubSubService.Publish(topic:= E_Topics.WORKING2_INBOUND_TOTE,data:= subData);
	A2	:= A2+1;
END_IF

//subData.Topic	:= E_Topics.RESET_WAITING_FOR_NEW_SPACE;
//GVL.PubSubService.Publish(topic:= E_Topics.RESET_WAITING_FOR_NEW_SPACE,data:= subData);
END_METHOD

{attribute 'TcRpcEnable'}
METHOD  init_tote_request : udint
VAR_INPUT
	init_tote_request_params : InitToteRequestParams;
END_VAR
init_tote_request:=1;
IF init_tote_request_params.source_id=ModelIdentifier.inbounding_position AND 
   init_tote_request_params.source_id=ModelIdentifier.working_position THEN 
  ;
     //MAIN.Machine.EM03.eState:=	E_WorkingStates.IDLE;				
//			MAIN.Machine.EM03.xLoading	:= FALSE;
//			MAIN.Machine.EM03.xUnloading	:= FALSE;
//			MAIN.Machine.EM03.xPerturbing := FALSE;
//			MAIN.Machine.EM03.xSwaping    := FALSE;
	 //MAIN.Machine.EM01.eState:=E_LoadingStates.IDLE;
END_IF  
IF init_tote_request_params.source_id=ModelIdentifier.working_position AND 
   init_tote_request_params.source_id=ModelIdentifier.outbound_position THEN 
;
    // MAIN.Machine.EM03.eState:=	E_WorkingStates.IDLE;				
//			MAIN.Machine.EM03.xLoading	:= FALSE;
//			MAIN.Machine.EM03.xUnloading	:= FALSE;
//			MAIN.Machine.EM03.xPerturbing := FALSE;
//			MAIN.Machine.EM03.xSwaping    := FALSE;
	// MAIN.Machine.EM04.eState:=E_UnloadingStates.IDLE;
END_IF  
init_tote_request:=0;
END_METHOD

METHOD M_mapping : BOOL
VAR_INPUT
END_VAR
END_METHOD

{attribute 'TcRpcEnable'}
METHOD outbound_tote_request : UDINT
VAR_INPUT
	outbound_tote_params : OutboundToteParams;	
END_VAR
VAR	
	subData	: PubSubData;
END_VAR
IF sInstanceName='tote_1' THEN
	IF NOT (GVL.fb_working1.xOutbound OR GVL.fb_working1.xInbound ) THEN//avoid cmd while outbounding
		subData.Topic	:= E_Topics.WORKING1_OUTBOUND_TOTE;
		GVL.PubSubService.Publish(topic:= E_Topics.WORKING1_OUTBOUND_TOTE,data:= subData);
	END_IF	
END_IF
IF sInstanceName='tote_2' THEN
	IF NOT (GVL.fb_working2.xOutbound OR GVL.fb_working2.xInbound ) THEN//avoid cmd while outbounding
		subData.Topic	:= E_Topics.WORKING2_OUTBOUND_TOTE;
		GVL.PubSubService.Publish(topic:= E_Topics.WORKING2_OUTBOUND_TOTE,data:= subData);
	END_IF
END_IF
END_METHOD

{attribute 'TcRpcEnable'}
METHOD perturb_tote_request : UDINT
VAR_INPUT
	perturb_tote_params : PerturbToteParams;	
END_VAR
IF //APP.Machine.CurrentStateEnum=E_PMLState.ePMLState_Execute 
//AND 
cmd=OrderToteCommand.DO_NOTHING
AND NOT MAIN.safety_1.bStop_button_unlock 
//AND NOT MAIN.safety_1.bBStop_button_unlock 
THEN
	cmd	:= OrderToteCommand.OPEN_BAG;
	perturb_tote_request:=0;
ELSE
	perturb_tote_request:=1;
END_IF
END_METHOD

{attribute 'TcRpcEnable'}
METHOD reset_tote_request : UDINT
VAR_INPUT
		
END_VAR
reset_tote_request	:= 1;

GVL.PackTags.Command.CntrlCmd:=1;

reset_tote_request	:= 0;
END_METHOD

{attribute 'TcRpcEnable'}
METHOD Setcmd : BOOL
VAR_INPUT
	orderToteCommand : OrderToteCommand;
END_VAR
cmd	:= orderToteCommand;
END_METHOD

{attribute 'TcRpcEnable'}
METHOD swap_tote_request : UDINT
VAR_INPUT
	swap_tote_params : SwapToteParams;	
END_VAR
IF //APP.Machine.CurrentStateEnum=E_PMLState.ePMLState_Execute 
//AND 
cmd=OrderToteCommand.DO_NOTHING
AND NOT MAIN.safety_1.bStop_button_unlock 
//AND NOT MAIN.safety_1.bBStop_button_unlock 
THEN
	cmd	:= OrderToteCommand.SWAP;
	swap_tote_request:=0;
ELSE
	swap_tote_request:=1;
END_IF
END_METHOD

END_FUNCTION_BLOCK

